// ---- DUTs/IO/PDOs/Outputs_B00B49A9.TcDUT
{attribute addProperty BoxType "EK1960-0000-0019"}
{attribute addProperty Id "Module_1_Channel_1_Standard_Output_X5_1AT %Q*BOOL811Module_1_Channel_2_Standard_Output_X5_2AT %Q*BOOL812Module_1_Channel_3_Standard_Output_X5_3AT %Q*BOOL813Module_1_Channel_4_Standard_Output_X5_4AT %Q*BOOL814Module_2_Channel_1_Standard_Output_X5_5AT %Q*BOOL811Module_2_Channel_2_Standard_Output_X5_6AT %Q*BOOL812Module_2_Channel_3_Standard_Output_X5_7AT %Q*BOOL813Module_2_Channel_4_Standard_Output_X5_8AT %Q*BOOL814Module_3_Channel_1_Standard_Output_X7_1AT %Q*BOOL811Module_3_Channel_2_Standard_Output_X7_2AT %Q*BOOL812Module_3_Channel_3_Standard_Output_X7_3AT %Q*BOOL813Module_3_Channel_4_Standard_Output_X7_4AT %Q*BOOL814Module_4_Channel_1_Standard_Output_X7_5AT %Q*BOOL811Module_4_Channel_2_Standard_Output_X7_6AT %Q*BOOL812Module_4_Channel_3_Standard_Output_X7_7AT %Q*BOOL813Module_4_Channel_4_Standard_Output_X7_8AT %Q*BOOL814Module_5_Channel_1_Standard_Output_X9_1AT %Q*BOOL811Module_5_Channel_2_Standard_Output_X9_2AT %Q*BOOL812Module_5_Channel_3_Standard_Output_X9_3AT %Q*BOOL813Module_5_Channel_4_Standard_Output_X9_4AT %Q*BOOL814Module_6_Channel_1_Standard_Output_X9_5AT %Q*BOOL811Module_6_Channel_2_Standard_Output_X9_6AT %Q*BOOL812Module_6_Channel_3_Standard_Output_X9_7AT %Q*BOOL813Module_6_Channel_4_Standard_Output_X9_8AT %Q*BOOL814Relais_Module_Channel_1_Standard_Output_X4_1_X4_5AT %Q*BOOL811Relais_Module_Channel_2_Standard_Output_X4_2_X4_6AT %Q*BOOL812Relais_Module_Channel_3_Standard_Output_X4_3_X4_7AT %Q*BOOL813Relais_Module_Channel_4_Standard_Output_X4_4_X4_8AT %Q*BOOL814"}
{attribute addProperty CRC "2953529769"}
{attribute addProperty SizeInBites "224"}
{attribute addProperty SizeInBytes "28"}
TYPE Outputs_B00B49A9 :
STRUCT
	{attribute addProperty Name "Module_1_Channel_1_Standard_Output_X5_1"}
	Module_1_Channel_1_Standard_Output_X5_1 AT %Q* : BOOL;
	{attribute addProperty Name "Module_1_Channel_2_Standard_Output_X5_2"}
	Module_1_Channel_2_Standard_Output_X5_2 AT %Q* : BOOL;
	{attribute addProperty Name "Module_1_Channel_3_Standard_Output_X5_3"}
	Module_1_Channel_3_Standard_Output_X5_3 AT %Q* : BOOL;
	{attribute addProperty Name "Module_1_Channel_4_Standard_Output_X5_4"}
	Module_1_Channel_4_Standard_Output_X5_4 AT %Q* : BOOL;
	{attribute addProperty Name "Module_2_Channel_1_Standard_Output_X5_5"}
	Module_2_Channel_1_Standard_Output_X5_5 AT %Q* : BOOL;
	{attribute addProperty Name "Module_2_Channel_2_Standard_Output_X5_6"}
	Module_2_Channel_2_Standard_Output_X5_6 AT %Q* : BOOL;
	{attribute addProperty Name "Module_2_Channel_3_Standard_Output_X5_7"}
	Module_2_Channel_3_Standard_Output_X5_7 AT %Q* : BOOL;
	{attribute addProperty Name "Module_2_Channel_4_Standard_Output_X5_8"}
	Module_2_Channel_4_Standard_Output_X5_8 AT %Q* : BOOL;
	{attribute addProperty Name "Module_3_Channel_1_Standard_Output_X7_1"}
	Module_3_Channel_1_Standard_Output_X7_1 AT %Q* : BOOL;
	{attribute addProperty Name "Module_3_Channel_2_Standard_Output_X7_2"}
	Module_3_Channel_2_Standard_Output_X7_2 AT %Q* : BOOL;
	{attribute addProperty Name "Module_3_Channel_3_Standard_Output_X7_3"}
	Module_3_Channel_3_Standard_Output_X7_3 AT %Q* : BOOL;
	{attribute addProperty Name "Module_3_Channel_4_Standard_Output_X7_4"}
	Module_3_Channel_4_Standard_Output_X7_4 AT %Q* : BOOL;
	{attribute addProperty Name "Module_4_Channel_1_Standard_Output_X7_5"}
	Module_4_Channel_1_Standard_Output_X7_5 AT %Q* : BOOL;
	{attribute addProperty Name "Module_4_Channel_2_Standard_Output_X7_6"}
	Module_4_Channel_2_Standard_Output_X7_6 AT %Q* : BOOL;
	{attribute addProperty Name "Module_4_Channel_3_Standard_Output_X7_7"}
	Module_4_Channel_3_Standard_Output_X7_7 AT %Q* : BOOL;
	{attribute addProperty Name "Module_4_Channel_4_Standard_Output_X7_8"}
	Module_4_Channel_4_Standard_Output_X7_8 AT %Q* : BOOL;
	{attribute addProperty Name "Module_5_Channel_1_Standard_Output_X9_1"}
	Module_5_Channel_1_Standard_Output_X9_1 AT %Q* : BOOL;
	{attribute addProperty Name "Module_5_Channel_2_Standard_Output_X9_2"}
	Module_5_Channel_2_Standard_Output_X9_2 AT %Q* : BOOL;
	{attribute addProperty Name "Module_5_Channel_3_Standard_Output_X9_3"}
	Module_5_Channel_3_Standard_Output_X9_3 AT %Q* : BOOL;
	{attribute addProperty Name "Module_5_Channel_4_Standard_Output_X9_4"}
	Module_5_Channel_4_Standard_Output_X9_4 AT %Q* : BOOL;
	{attribute addProperty Name "Module_6_Channel_1_Standard_Output_X9_5"}
	Module_6_Channel_1_Standard_Output_X9_5 AT %Q* : BOOL;
	{attribute addProperty Name "Module_6_Channel_2_Standard_Output_X9_6"}
	Module_6_Channel_2_Standard_Output_X9_6 AT %Q* : BOOL;
	{attribute addProperty Name "Module_6_Channel_3_Standard_Output_X9_7"}
	Module_6_Channel_3_Standard_Output_X9_7 AT %Q* : BOOL;
	{attribute addProperty Name "Module_6_Channel_4_Standard_Output_X9_8"}
	Module_6_Channel_4_Standard_Output_X9_8 AT %Q* : BOOL;
	{attribute addProperty Name "Relais_Module_Channel_1_Standard_Output_X4_1_X4_5"}
	Relais_Module_Channel_1_Standard_Output_X4_1_X4_5 AT %Q* : BOOL;
	{attribute addProperty Name "Relais_Module_Channel_2_Standard_Output_X4_2_X4_6"}
	Relais_Module_Channel_2_Standard_Output_X4_2_X4_6 AT %Q* : BOOL;
	{attribute addProperty Name "Relais_Module_Channel_3_Standard_Output_X4_3_X4_7"}
	Relais_Module_Channel_3_Standard_Output_X4_3_X4_7 AT %Q* : BOOL;
	{attribute addProperty Name "Relais_Module_Channel_4_Standard_Output_X4_4_X4_8"}
	Relais_Module_Channel_4_Standard_Output_X4_4_X4_8 AT %Q* : BOOL;
END_STRUCT
END_TYPE

// ---- DUTs/IO/PDOs/Module_1_FSoE_DD00D81F.TcDUT
{attribute addProperty BoxType "EK1960-0000-0019"}
{attribute addProperty Id "FSoE_InputsFSoE_Inputs_FED5CD6512015FSoE_OutputsFSoE_Outputs_931DC9C512015"}
{attribute addProperty CRC "3707820063"}
{attribute addProperty SizeInBites "240"}
{attribute addProperty SizeInBytes "30"}
TYPE Module_1_FSoE_DD00D81F :
STRUCT
	{attribute addProperty Name "FSoE_Inputs"}
	FSoE_Inputs  : FSoE_Inputs_FED5CD65;
	{attribute addProperty Name "FSoE_Outputs"}
	FSoE_Outputs  : FSoE_Outputs_931DC9C5;
END_STRUCT
END_TYPE

// ---- DUTs/IO/PDOs/Module_2_FSOUT_3AD10D8E.TcDUT
{attribute addProperty BoxType "EK1960-0000-0019"}
{attribute addProperty Id "OutputsOutputs_B00B49A922428"}
{attribute addProperty CRC "986779022"}
{attribute addProperty SizeInBites "224"}
{attribute addProperty SizeInBytes "28"}
TYPE Module_2_FSOUT_3AD10D8E :
STRUCT
	{attribute addProperty Name "Outputs"}
	Outputs  : Outputs_B00B49A9;
END_STRUCT
END_TYPE

// ---- DUTs/IO/PDOs/FSoE_Inputs_91F6EA71.TcDUT
{attribute addProperty BoxType "EK1960-0000-0021"}
{attribute addProperty Id "FSOEAT %I*FSOE_320A0AF812015"}
{attribute addProperty CRC "2448878193"}
{attribute addProperty SizeInBites "120"}
{attribute addProperty SizeInBytes "15"}
TYPE FSoE_Inputs_91F6EA71 :
STRUCT
	{attribute addProperty Name "FSOE"}
	FSOE AT %I* : FSOE_320A0AF8;
END_STRUCT
END_TYPE

// ---- DUTs/IO/PDOs/FSoE_Outputs_DB0FA8F7.TcDUT
{attribute addProperty BoxType "EK1960-0000-0021"}
{attribute addProperty Id "FSOEAT %Q*FSOE_B358BD5C12015"}
{attribute addProperty CRC "3675236599"}
{attribute addProperty SizeInBites "120"}
{attribute addProperty SizeInBytes "15"}
TYPE FSoE_Outputs_DB0FA8F7 :
STRUCT
	{attribute addProperty Name "FSOE"}
	FSOE AT %Q* : FSOE_B358BD5C;
END_STRUCT
END_TYPE

// ---- DUTs/IO/PDOs/Outputs_5BA3BA9A.TcDUT
{attribute addProperty BoxType "EK1960-0000-0021"}
{attribute addProperty Id "Module_1_Channel_1_Standard_Output_X5_1AT %Q*BOOL811Module_1_Channel_2_Standard_Output_X5_2AT %Q*BOOL812Module_1_Channel_3_Standard_Output_X5_3AT %Q*BOOL813Module_1_Channel_4_Standard_Output_X5_4AT %Q*BOOL814Module_2_Channel_1_Standard_Output_X5_5AT %Q*BOOL811Module_2_Channel_2_Standard_Output_X5_6AT %Q*BOOL812Module_2_Channel_3_Standard_Output_X5_7AT %Q*BOOL813Module_2_Channel_4_Standard_Output_X5_8AT %Q*BOOL814Module_3_Channel_1_Standard_Output_X7_1AT %Q*BOOL811Module_3_Channel_2_Standard_Output_X7_2AT %Q*BOOL812Module_3_Channel_3_Standard_Output_X7_3AT %Q*BOOL813Module_3_Channel_4_Standard_Output_X7_4AT %Q*BOOL814Module_4_Channel_1_Standard_Output_X7_5AT %Q*BOOL811Module_4_Channel_2_Standard_Output_X7_6AT %Q*BOOL812Module_4_Channel_3_Standard_Output_X7_7AT %Q*BOOL813Module_4_Channel_4_Standard_Output_X7_8AT %Q*BOOL814Module_5_Channel_1_Standard_Output_X9_1AT %Q*BOOL811Module_5_Channel_2_Standard_Output_X9_2AT %Q*BOOL812Module_5_Channel_3_Standard_Output_X9_3AT %Q*BOOL813Module_5_Channel_4_Standard_Output_X9_4AT %Q*BOOL814Module_6_Channel_1_Standard_Output_X9_5AT %Q*BOOL811Module_6_Channel_2_Standard_Output_X9_6AT %Q*BOOL812Module_6_Channel_3_Standard_Output_X9_7AT %Q*BOOL813Module_6_Channel_4_Standard_Output_X9_8AT %Q*BOOL814"}
{attribute addProperty CRC "1537456794"}
{attribute addProperty SizeInBites "192"}
{attribute addProperty SizeInBytes "24"}
TYPE Outputs_5BA3BA9A :
STRUCT
	{attribute addProperty Name "Module_1_Channel_1_Standard_Output_X5_1"}
	Module_1_Channel_1_Standard_Output_X5_1 AT %Q* : BOOL;
	{attribute addProperty Name "Module_1_Channel_2_Standard_Output_X5_2"}
	Module_1_Channel_2_Standard_Output_X5_2 AT %Q* : BOOL;
	{attribute addProperty Name "Module_1_Channel_3_Standard_Output_X5_3"}
	Module_1_Channel_3_Standard_Output_X5_3 AT %Q* : BOOL;
	{attribute addProperty Name "Module_1_Channel_4_Standard_Output_X5_4"}
	Module_1_Channel_4_Standard_Output_X5_4 AT %Q* : BOOL;
	{attribute addProperty Name "Module_2_Channel_1_Standard_Output_X5_5"}
	Module_2_Channel_1_Standard_Output_X5_5 AT %Q* : BOOL;
	{attribute addProperty Name "Module_2_Channel_2_Standard_Output_X5_6"}
	Module_2_Channel_2_Standard_Output_X5_6 AT %Q* : BOOL;
	{attribute addProperty Name "Module_2_Channel_3_Standard_Output_X5_7"}
	Module_2_Channel_3_Standard_Output_X5_7 AT %Q* : BOOL;
	{attribute addProperty Name "Module_2_Channel_4_Standard_Output_X5_8"}
	Module_2_Channel_4_Standard_Output_X5_8 AT %Q* : BOOL;
	{attribute addProperty Name "Module_3_Channel_1_Standard_Output_X7_1"}
	Module_3_Channel_1_Standard_Output_X7_1 AT %Q* : BOOL;
	{attribute addProperty Name "Module_3_Channel_2_Standard_Output_X7_2"}
	Module_3_Channel_2_Standard_Output_X7_2 AT %Q* : BOOL;
	{attribute addProperty Name "Module_3_Channel_3_Standard_Output_X7_3"}
	Module_3_Channel_3_Standard_Output_X7_3 AT %Q* : BOOL;
	{attribute addProperty Name "Module_3_Channel_4_Standard_Output_X7_4"}
	Module_3_Channel_4_Standard_Output_X7_4 AT %Q* : BOOL;
	{attribute addProperty Name "Module_4_Channel_1_Standard_Output_X7_5"}
	Module_4_Channel_1_Standard_Output_X7_5 AT %Q* : BOOL;
	{attribute addProperty Name "Module_4_Channel_2_Standard_Output_X7_6"}
	Module_4_Channel_2_Standard_Output_X7_6 AT %Q* : BOOL;
	{attribute addProperty Name "Module_4_Channel_3_Standard_Output_X7_7"}
	Module_4_Channel_3_Standard_Output_X7_7 AT %Q* : BOOL;
	{attribute addProperty Name "Module_4_Channel_4_Standard_Output_X7_8"}
	Module_4_Channel_4_Standard_Output_X7_8 AT %Q* : BOOL;
	{attribute addProperty Name "Module_5_Channel_1_Standard_Output_X9_1"}
	Module_5_Channel_1_Standard_Output_X9_1 AT %Q* : BOOL;
	{attribute addProperty Name "Module_5_Channel_2_Standard_Output_X9_2"}
	Module_5_Channel_2_Standard_Output_X9_2 AT %Q* : BOOL;
	{attribute addProperty Name "Module_5_Channel_3_Standard_Output_X9_3"}
	Module_5_Channel_3_Standard_Output_X9_3 AT %Q* : BOOL;
	{attribute addProperty Name "Module_5_Channel_4_Standard_Output_X9_4"}
	Module_5_Channel_4_Standard_Output_X9_4 AT %Q* : BOOL;
	{attribute addProperty Name "Module_6_Channel_1_Standard_Output_X9_5"}
	Module_6_Channel_1_Standard_Output_X9_5 AT %Q* : BOOL;
	{attribute addProperty Name "Module_6_Channel_2_Standard_Output_X9_6"}
	Module_6_Channel_2_Standard_Output_X9_6 AT %Q* : BOOL;
	{attribute addProperty Name "Module_6_Channel_3_Standard_Output_X9_7"}
	Module_6_Channel_3_Standard_Output_X9_7 AT %Q* : BOOL;
	{attribute addProperty Name "Module_6_Channel_4_Standard_Output_X9_8"}
	Module_6_Channel_4_Standard_Output_X9_8 AT %Q* : BOOL;
END_STRUCT
END_TYPE

// ---- DUTs/IO/PDOs/Module_1_FSoE_DA01C73E.TcDUT
{attribute addProperty BoxType "EK1960-0000-0021"}
{attribute addProperty Id "FSoE_InputsFSoE_Inputs_91F6EA7112015FSoE_OutputsFSoE_Outputs_DB0FA8F712015"}
{attribute addProperty CRC "3657549630"}
{attribute addProperty SizeInBites "240"}
{attribute addProperty SizeInBytes "30"}
TYPE Module_1_FSoE_DA01C73E :
STRUCT
	{attribute addProperty Name "FSoE_Inputs"}
	FSoE_Inputs  : FSoE_Inputs_91F6EA71;
	{attribute addProperty Name "FSoE_Outputs"}
	FSoE_Outputs  : FSoE_Outputs_DB0FA8F7;
END_STRUCT
END_TYPE

// ---- DUTs/IO/PDOs/Module_2_FSOUT_9F3624CE.TcDUT
{attribute addProperty BoxType "EK1960-0000-0021"}
{attribute addProperty Id "OutputsOutputs_5BA3BA9A19224"}
{attribute addProperty CRC "2671125710"}
{attribute addProperty SizeInBites "192"}
{attribute addProperty SizeInBytes "24"}
TYPE Module_2_FSOUT_9F3624CE :
STRUCT
	{attribute addProperty Name "Outputs"}
	Outputs  : Outputs_5BA3BA9A;
END_STRUCT
END_TYPE

// ---- DUTs/IO/PDOs/FSoE_Inputs_0C161FF7.TcDUT
{attribute addProperty BoxType "EK1960-2600-0019"}
{attribute addProperty Id "FSOEAT %I*FSOE_704ED52312015"}
{attribute addProperty CRC "202776567"}
{attribute addProperty SizeInBites "120"}
{attribute addProperty SizeInBytes "15"}
TYPE FSoE_Inputs_0C161FF7 :
STRUCT
	{attribute addProperty Name "FSOE"}
	FSOE AT %I* : FSOE_704ED523;
END_STRUCT
END_TYPE

// ---- DUTs/IO/PDOs/FSoE_Outputs_E86FAAD6.TcDUT
{attribute addProperty BoxType "EK1960-2600-0019"}
{attribute addProperty Id "FSOEAT %Q*FSOE_340991D312015"}
{attribute addProperty CRC "3899632342"}
{attribute addProperty SizeInBites "120"}
{attribute addProperty SizeInBytes "15"}
TYPE FSoE_Outputs_E86FAAD6 :
STRUCT
	{attribute addProperty Name "FSOE"}
	FSOE AT %Q* : FSOE_340991D3;
END_STRUCT
END_TYPE

// ---- DUTs/IO/PDOs/Module_1_FSoE_DA1FCD51.TcDUT
{attribute addProperty BoxType "EK1960-2600-0019"}
{attribute addProperty Id "FSoE_InputsFSoE_Inputs_0C161FF712015FSoE_OutputsFSoE_Outputs_E86FAAD612015"}
{attribute addProperty CRC "3659517265"}
{attribute addProperty SizeInBites "240"}
{attribute addProperty SizeInBytes "30"}
TYPE Module_1_FSoE_DA1FCD51 :
STRUCT
	{attribute addProperty Name "FSoE_Inputs"}
	FSoE_Inputs  : FSoE_Inputs_0C161FF7;
	{attribute addProperty Name "FSoE_Outputs"}
	FSoE_Outputs  : FSoE_Outputs_E86FAAD6;
END_STRUCT
END_TYPE

// ---- DUTs/IO/PDOs/FSoE_Inputs_CBB11F24.TcDUT
{attribute addProperty BoxType "EK1960-2600-0021"}
{attribute addProperty Id "FSOEAT %I*FSOE_3B47B0C112015"}
{attribute addProperty CRC "3417382692"}
{attribute addProperty SizeInBites "120"}
{attribute addProperty SizeInBytes "15"}
TYPE FSoE_Inputs_CBB11F24 :
STRUCT
	{attribute addProperty Name "FSOE"}
	FSOE AT %I* : FSOE_3B47B0C1;
END_STRUCT
END_TYPE

// ---- DUTs/IO/PDOs/FSoE_Outputs_616B4B11.TcDUT
{attribute addProperty BoxType "EK1960-2600-0021"}
{attribute addProperty Id "FSOEAT %Q*FSOE_9F05737212015"}
{attribute addProperty CRC "1634421521"}
{attribute addProperty SizeInBites "120"}
{attribute addProperty SizeInBytes "15"}
TYPE FSoE_Outputs_616B4B11 :
STRUCT
	{attribute addProperty Name "FSOE"}
	FSOE AT %Q* : FSOE_9F057372;
END_STRUCT
END_TYPE

// ---- DUTs/IO/PDOs/Module_1_FSoE_1C2EAE46.TcDUT
{attribute addProperty BoxType "EK1960-2600-0021"}
{attribute addProperty Id "FSoE_InputsFSoE_Inputs_CBB11F2412015FSoE_OutputsFSoE_Outputs_616B4B1112015"}
{attribute addProperty CRC "472821318"}
{attribute addProperty SizeInBites "240"}
{attribute addProperty SizeInBytes "30"}
TYPE Module_1_FSoE_1C2EAE46 :
STRUCT
	{attribute addProperty Name "FSoE_Inputs"}
	FSoE_Inputs  : FSoE_Inputs_CBB11F24;
	{attribute addProperty Name "FSoE_Outputs"}
	FSoE_Outputs  : FSoE_Outputs_616B4B11;
END_STRUCT
END_TYPE

// ---- DUTs/IO/Boxes/EK1100_179A0949.TcDUT
{attribute addProperty BoxType "EK1100-0000-0018"}
{attribute addProperty Id "InfoDataInfoData_192954DE162"}
{attribute addProperty CRC "395970889"}
{attribute addProperty SizeInBites "16"}
{attribute addProperty SizeInBytes "2"}
TYPE EK1100_179A0949 :
STRUCT
	{attribute addProperty Name "InfoData"}
	InfoData : InfoData_192954DE;
END_STRUCT
END_TYPE

// ---- DUTs/IO/Boxes/EK1122_179A0949.TcDUT
{attribute addProperty BoxType "EK1122-0000-0018"}
{attribute addProperty Id "InfoDataInfoData_192954DE162"}
{attribute addProperty CRC "395970889"}
{attribute addProperty SizeInBites "16"}
{attribute addProperty SizeInBytes "2"}
TYPE EK1122_179A0949 :
STRUCT
	{attribute addProperty Name "InfoData"}
	InfoData : InfoData_192954DE;
END_STRUCT
END_TYPE

// ---- DUTs/IO/Boxes/EJ1100_179A0949.TcDUT
{attribute addProperty BoxType "EJ1100-0000-0018"}
{attribute addProperty Id "InfoDataInfoData_192954DE162"}
{attribute addProperty CRC "395970889"}
{attribute addProperty SizeInBites "16"}
{attribute addProperty SizeInBytes "2"}
TYPE EJ1100_179A0949 :
STRUCT
	{attribute addProperty Name "InfoData"}
	InfoData : InfoData_192954DE;
END_STRUCT
END_TYPE

// ---- DUTs/IO/Boxes/EJ1101_6969C224.TcDUT
{attribute addProperty BoxType "EJ1101-0022-0016"}
{attribute addProperty Id "WcStateAT %I*WcState_28A8677510.1250InfoDataAT %I*InfoData_BC63D37F80100"}
{attribute addProperty CRC "752626490"}
{attribute addProperty SizeInBites "81"}
{attribute addProperty SizeInBytes "10.125"}
TYPE EJ1101_6969C224 :
STRUCT
	{attribute addProperty Name "WcState"}
	WcState : WcState_28A86775;
	{attribute addProperty Name "InfoData"}
	InfoData : InfoData_BC63D37F;
END_STRUCT
END_TYPE

// ---- DUTs/IO/Boxes/EJ1008_772BB414.TcDUT
{attribute addProperty BoxType "EJ1008-0000-0017"}
{attribute addProperty Id "ChannelAT %I*ARRAY[0..7] OF Channel_E4AEF59E6480WcStateAT %I*WcState_98A4DF7520.250InfoDataAT %I*InfoData_192954DE1620"}
{attribute addProperty CRC "2007808796"}
{attribute addProperty SizeInBites "82"}
{attribute addProperty SizeInBytes "10.25"}
TYPE EJ1008_772BB414 :
STRUCT
	{attribute addProperty Name "Channel"}
	Channel : ARRAY[0..7] OF Channel_E4AEF59E;
	{attribute addProperty Name "WcState"}
	WcState : WcState_98A4DF75;
	{attribute addProperty Name "InfoData"}
	InfoData : InfoData_192954DE;
END_STRUCT
END_TYPE

// ---- DUTs/IO/Boxes/EJ1128_772BB414.TcDUT
{attribute addProperty BoxType "EJ1128-0000-0016"}
{attribute addProperty Id "ChannelAT %I*ARRAY[0..7] OF Channel_E4AEF59E6480WcStateAT %I*WcState_98A4DF7520.250InfoDataAT %I*InfoData_192954DE1620"}
{attribute addProperty CRC "2007808796"}
{attribute addProperty SizeInBites "82"}
{attribute addProperty SizeInBytes "10.25"}
TYPE EJ1128_772BB414 :
STRUCT
	{attribute addProperty Name "Channel"}
	Channel : ARRAY[0..7] OF Channel_E4AEF59E;
	{attribute addProperty Name "WcState"}
	WcState : WcState_98A4DF75;
	{attribute addProperty Name "InfoData"}
	InfoData : InfoData_192954DE;
END_STRUCT
END_TYPE

// ---- DUTs/IO/Boxes/EJ1809_248EAA34.TcDUT
{attribute addProperty BoxType "EJ1809-0000-0017"}
{attribute addProperty Id "ChannelAT %I*ARRAY[0..15] OF Channel_E4AEF59E128160WcStateAT %I*WcState_98A4DF7520.250InfoDataAT %I*InfoData_192954DE1620"}
{attribute addProperty CRC "4206052659"}
{attribute addProperty SizeInBites "146"}
{attribute addProperty SizeInBytes "18.25"}
TYPE EJ1809_248EAA34 :
STRUCT
	{attribute addProperty Name "Channel"}
	Channel : ARRAY[0..15] OF Channel_E4AEF59E;
	{attribute addProperty Name "WcState"}
	WcState : WcState_98A4DF75;
	{attribute addProperty Name "InfoData"}
	InfoData : InfoData_192954DE;
END_STRUCT
END_TYPE

// ---- DUTs/IO/Boxes/EJ1819_248EAA34.TcDUT
{attribute addProperty BoxType "EJ1819-0000-0017"}
{attribute addProperty Id "ChannelAT %I*ARRAY[0..15] OF Channel_E4AEF59E128160WcStateAT %I*WcState_98A4DF7520.250InfoDataAT %I*InfoData_192954DE1620"}
{attribute addProperty CRC "4206052659"}
{attribute addProperty SizeInBites "146"}
{attribute addProperty SizeInBytes "18.25"}
TYPE EJ1819_248EAA34 :
STRUCT
	{attribute addProperty Name "Channel"}
	Channel : ARRAY[0..15] OF Channel_E4AEF59E;
	{attribute addProperty Name "WcState"}
	WcState : WcState_98A4DF75;
	{attribute addProperty Name "InfoData"}
	InfoData : InfoData_192954DE;
END_STRUCT
END_TYPE

// ---- DUTs/IO/Boxes/EJ1859_538B459D.TcDUT
{attribute addProperty BoxType "EJ1859-0000-0017"}
{attribute addProperty Id "ChannelAT %I*ARRAY[0..7] OF Channel_E4AEF59E6480Channel_1AT %Q*ARRAY[0..7] OF Channel_7F374EB06480WcStateAT %I*WcState_98A4DF7520.250InfoDataAT %I*InfoData_192954DE1620"}
{attribute addProperty CRC "4038043443"}
{attribute addProperty SizeInBites "146"}
{attribute addProperty SizeInBytes "18.25"}
TYPE EJ1859_538B459D :
STRUCT
	{attribute addProperty Name "Channel"}
	Channel : ARRAY[0..7] OF Channel_E4AEF59E;
	{attribute addProperty Name "Channel_1"}
	Channel_1 : ARRAY[0..7] OF Channel_7F374EB0;
	{attribute addProperty Name "WcState"}
	WcState : WcState_98A4DF75;
	{attribute addProperty Name "InfoData"}
	InfoData : InfoData_192954DE;
END_STRUCT
END_TYPE

// ---- DUTs/IO/Boxes/EJ1889_248EAA34.TcDUT
{attribute addProperty BoxType "EJ1889-0000-0017"}
{attribute addProperty Id "ChannelAT %I*ARRAY[0..15] OF Channel_E4AEF59E128160WcStateAT %I*WcState_98A4DF7520.250InfoDataAT %I*InfoData_192954DE1620"}
{attribute addProperty CRC "4206052659"}
{attribute addProperty SizeInBites "146"}
{attribute addProperty SizeInBytes "18.25"}
TYPE EJ1889_248EAA34 :
STRUCT
	{attribute addProperty Name "Channel"}
	Channel : ARRAY[0..15] OF Channel_E4AEF59E;
	{attribute addProperty Name "WcState"}
	WcState : WcState_98A4DF75;
	{attribute addProperty Name "InfoData"}
	InfoData : InfoData_192954DE;
END_STRUCT
END_TYPE

// ---- DUTs/IO/Boxes/EJ1122_179A0949.TcDUT
{attribute addProperty BoxType "EJ1122-0000-0016"}
{attribute addProperty Id "InfoDataInfoData_192954DE162"}
{attribute addProperty CRC "395970889"}
{attribute addProperty SizeInBites "16"}
{attribute addProperty SizeInBytes "2"}
TYPE EJ1122_179A0949 :
STRUCT
	{attribute addProperty Name "InfoData"}
	InfoData : InfoData_192954DE;
END_STRUCT
END_TYPE

// ---- DUTs/IO/Boxes/EJ2008_A854BE6D.TcDUT
{attribute addProperty BoxType "EJ2008-0000-0017"}
{attribute addProperty Id "ChannelAT %Q*ARRAY[0..7] OF Channel_7F374EB06480WcStateAT %I*WcState_28A8677510.1250InfoDataAT %I*InfoData_192954DE1620"}
{attribute addProperty CRC "1482585628"}
{attribute addProperty SizeInBites "81"}
{attribute addProperty SizeInBytes "10.125"}
TYPE EJ2008_A854BE6D :
STRUCT
	{attribute addProperty Name "Channel"}
	Channel : ARRAY[0..7] OF Channel_7F374EB0;
	{attribute addProperty Name "WcState"}
	WcState : WcState_28A86775;
	{attribute addProperty Name "InfoData"}
	InfoData : InfoData_192954DE;
END_STRUCT
END_TYPE

// ---- DUTs/IO/Boxes/EJ2128_A854BE6D.TcDUT
{attribute addProperty BoxType "EJ2128-0000-0016"}
{attribute addProperty Id "ChannelAT %Q*ARRAY[0..7] OF Channel_7F374EB06480WcStateAT %I*WcState_28A8677510.1250InfoDataAT %I*InfoData_192954DE1620"}
{attribute addProperty CRC "1482585628"}
{attribute addProperty SizeInBites "81"}
{attribute addProperty SizeInBytes "10.125"}
TYPE EJ2128_A854BE6D :
STRUCT
	{attribute addProperty Name "Channel"}
	Channel : ARRAY[0..7] OF Channel_7F374EB0;
	{attribute addProperty Name "WcState"}
	WcState : WcState_28A86775;
	{attribute addProperty Name "InfoData"}
	InfoData : InfoData_192954DE;
END_STRUCT
END_TYPE

// ---- DUTs/IO/Boxes/EJ2502_68F74D5A.TcDUT
{attribute addProperty BoxType "EJ2502-0000-0023"}
{attribute addProperty Id "PWM_Outputs_ChannelAT %Q*ARRAY[0..1] OF PWM_Outputs_Channel_A83D42AA3240WcStateAT %I*WcState_28A8677510.1250InfoDataAT %I*InfoData_BC63D37F80100"}
{attribute addProperty CRC "1493002450"}
{attribute addProperty SizeInBites "113"}
{attribute addProperty SizeInBytes "14.125"}
TYPE EJ2502_68F74D5A :
STRUCT
	{attribute addProperty Name "PWM_Outputs_Channel"}
	PWM_Outputs_Channel : ARRAY[0..1] OF PWM_Outputs_Channel_A83D42AA;
	{attribute addProperty Name "WcState"}
	WcState : WcState_28A86775;
	{attribute addProperty Name "InfoData"}
	InfoData : InfoData_BC63D37F;
END_STRUCT
END_TYPE

// ---- DUTs/IO/Boxes/EJ2521_A10F5EEB.TcDUT
{attribute addProperty BoxType "EJ2521-0224-0016"}
{attribute addProperty Id "PTO_StatusAT %I*PTO_Status_B9BB57FE1620ENC_Status_compactAT %I*ENC_Status_compact_FA080ECA4860PLS_Status_ChannelAT %I*ARRAY[0..1] OF PLS_Status_Channel_7A2392D13240PTO_ControlAT %Q*PTO_Control_0A6210C33240PTO_Target_compactAT %Q*PTO_Target_compact_C80C22BB1620ENC_Control_compactAT %Q*ENC_Control_compact_5C86AA9D3240PLS_Control_compact_ChannelAT %Q*ARRAY[0..3] OF PLS_Control_compact_Channel_F7E9C67496120WcStateAT %I*WcState_98A4DF7520.250InfoDataAT %I*InfoData_BC63D37F80100"}
{attribute addProperty CRC "3307808944"}
{attribute addProperty SizeInBites "354"}
{attribute addProperty SizeInBytes "44.25"}
TYPE EJ2521_A10F5EEB :
STRUCT
	{attribute addProperty Name "PTO_Status"}
	PTO_Status : PTO_Status_B9BB57FE;
	{attribute addProperty Name "ENC_Status_compact"}
	ENC_Status_compact : ENC_Status_compact_FA080ECA;
	{attribute addProperty Name "PLS_Status_Channel"}
	PLS_Status_Channel : ARRAY[0..1] OF PLS_Status_Channel_7A2392D1;
	{attribute addProperty Name "PTO_Control"}
	PTO_Control : PTO_Control_0A6210C3;
	{attribute addProperty Name "PTO_Target_compact"}
	PTO_Target_compact : PTO_Target_compact_C80C22BB;
	{attribute addProperty Name "ENC_Control_compact"}
	ENC_Control_compact : ENC_Control_compact_5C86AA9D;
	{attribute addProperty Name "PLS_Control_compact_Channel"}
	PLS_Control_compact_Channel : ARRAY[0..3] OF PLS_Control_compact_Channel_F7E9C674;
	{attribute addProperty Name "WcState"}
	WcState : WcState_98A4DF75;
	{attribute addProperty Name "InfoData"}
	InfoData : InfoData_BC63D37F;
END_STRUCT
END_TYPE

// ---- DUTs/IO/Boxes/EJ2522_58A1BC1F.TcDUT
{attribute addProperty BoxType "EJ2522-0000-0022"}
{attribute addProperty Id "PTO_Status_ChannelAT %I*ARRAY[0..1] OF PTO_Status_Channel_B9BB57FE3240ENC_Status_ChannelAT %I*ARRAY[0..2] OF ENC_Status_Channel_D7F8917396120PTO_Control_Channel_1AT %Q*PTO_Control_Channel_0A6210C33240PTO_Target_Channel_1AT %Q*PTO_Target_Channel_3945899C3240PTO_Control_Channel_2AT %Q*PTO_Control_Channel_0A6210C33240PTO_Target_Channel_2AT %Q*PTO_Target_Channel_3945899C3240ENC_Control_ChannelAT %Q*ARRAY[0..2] OF ENC_Control_Channel_8309D56E96120WcStateAT %I*WcState_98A4DF7520.250InfoDataAT %I*InfoData_BC63D37F80100"}
{attribute addProperty CRC "1184876195"}
{attribute addProperty SizeInBites "434"}
{attribute addProperty SizeInBytes "54.25"}
TYPE EJ2522_58A1BC1F :
STRUCT
	{attribute addProperty Name "PTO_Status_Channel"}
	PTO_Status_Channel : ARRAY[0..1] OF PTO_Status_Channel_B9BB57FE;
	{attribute addProperty Name "ENC_Status_Channel"}
	ENC_Status_Channel : ARRAY[0..2] OF ENC_Status_Channel_D7F89173;
	{attribute addProperty Name "PTO_Control_Channel_1"}
	PTO_Control_Channel_1 : PTO_Control_Channel_0A6210C3;
	{attribute addProperty Name "PTO_Target_Channel_1"}
	PTO_Target_Channel_1 : PTO_Target_Channel_3945899C;
	{attribute addProperty Name "PTO_Control_Channel_2"}
	PTO_Control_Channel_2 : PTO_Control_Channel_0A6210C3;
	{attribute addProperty Name "PTO_Target_Channel_2"}
	PTO_Target_Channel_2 : PTO_Target_Channel_3945899C;
	{attribute addProperty Name "ENC_Control_Channel"}
	ENC_Control_Channel : ARRAY[0..2] OF ENC_Control_Channel_8309D56E;
	{attribute addProperty Name "WcState"}
	WcState : WcState_98A4DF75;
	{attribute addProperty Name "InfoData"}
	InfoData : InfoData_BC63D37F;
END_STRUCT
END_TYPE

// ---- DUTs/IO/Boxes/EJ2809_859F43D2.TcDUT
{attribute addProperty BoxType "EJ2809-0000-0017"}
{attribute addProperty Id "ChannelAT %Q*ARRAY[0..15] OF Channel_7F374EB0128160WcStateAT %I*WcState_28A8677510.1250InfoDataAT %I*InfoData_192954DE1620"}
{attribute addProperty CRC "924279498"}
{attribute addProperty SizeInBites "145"}
{attribute addProperty SizeInBytes "18.125"}
TYPE EJ2809_859F43D2 :
STRUCT
	{attribute addProperty Name "Channel"}
	Channel : ARRAY[0..15] OF Channel_7F374EB0;
	{attribute addProperty Name "WcState"}
	WcState : WcState_28A86775;
	{attribute addProperty Name "InfoData"}
	InfoData : InfoData_192954DE;
END_STRUCT
END_TYPE

// ---- DUTs/IO/Boxes/EJ2889_859F43D2.TcDUT
{attribute addProperty BoxType "EJ2889-0000-0016"}
{attribute addProperty Id "ChannelAT %Q*ARRAY[0..15] OF Channel_7F374EB0128160WcStateAT %I*WcState_28A8677510.1250InfoDataAT %I*InfoData_192954DE1620"}
{attribute addProperty CRC "924279498"}
{attribute addProperty SizeInBites "145"}
{attribute addProperty SizeInBytes "18.125"}
TYPE EJ2889_859F43D2 :
STRUCT
	{attribute addProperty Name "Channel"}
	Channel : ARRAY[0..15] OF Channel_7F374EB0;
	{attribute addProperty Name "WcState"}
	WcState : WcState_28A86775;
	{attribute addProperty Name "InfoData"}
	InfoData : InfoData_192954DE;
END_STRUCT
END_TYPE

// ---- DUTs/IO/Boxes/EJ3004_25122C20.TcDUT
{attribute addProperty BoxType "EJ3004-0000-0019"}
{attribute addProperty Id "AI_Standard_ChannelAT %I*ARRAY[0..6] OF AI_Standard_Channel_5763EEB9128160WcStateAT %I*WcState_98A4DF7520.250InfoDataAT %I*InfoData_BC63D37F80100"}
{attribute addProperty CRC "3504630615"}
{attribute addProperty SizeInBites "210"}
{attribute addProperty SizeInBytes "26.25"}
TYPE EJ3004_25122C20 :
STRUCT
	{attribute addProperty Name "AI_Standard_Channel"}
	AI_Standard_Channel : ARRAY[0..6] OF AI_Standard_Channel_5763EEB9;
	{attribute addProperty Name "WcState"}
	WcState : WcState_98A4DF75;
	{attribute addProperty Name "InfoData"}
	InfoData : InfoData_BC63D37F;
END_STRUCT
END_TYPE

// ---- DUTs/IO/Boxes/EJ3004_BB821456.TcDUT
{attribute addProperty BoxType "EJ3004-0000-0020"}
{attribute addProperty Id "AI_Standard_ChannelAT %I*ARRAY[0..6] OF AI_Standard_Channel_F16A160D128160WcStateAT %I*WcState_98A4DF7520.250InfoDataAT %I*InfoData_BC63D37F80100"}
{attribute addProperty CRC "4042565249"}
{attribute addProperty SizeInBites "210"}
{attribute addProperty SizeInBytes "26.25"}
TYPE EJ3004_BB821456 :
STRUCT
	{attribute addProperty Name "AI_Standard_Channel"}
	AI_Standard_Channel : ARRAY[0..6] OF AI_Standard_Channel_F16A160D;
	{attribute addProperty Name "WcState"}
	WcState : WcState_98A4DF75;
	{attribute addProperty Name "InfoData"}
	InfoData : InfoData_BC63D37F;
END_STRUCT
END_TYPE

// ---- DUTs/IO/Boxes/EJ3048_EA60A077.TcDUT
{attribute addProperty BoxType "EJ3048-0000-0020"}
{attribute addProperty Id "AI_Standard_ChannelAT %I*ARRAY[0..14] OF AI_Standard_Channel_F16A160D256320WcStateAT %I*WcState_98A4DF7520.250InfoDataAT %I*InfoData_BC63D37F80100"}
{attribute addProperty CRC "1252681791"}
{attribute addProperty SizeInBites "338"}
{attribute addProperty SizeInBytes "42.25"}
TYPE EJ3048_EA60A077 :
STRUCT
	{attribute addProperty Name "AI_Standard_Channel"}
	AI_Standard_Channel : ARRAY[0..14] OF AI_Standard_Channel_F16A160D;
	{attribute addProperty Name "WcState"}
	WcState : WcState_98A4DF75;
	{attribute addProperty Name "InfoData"}
	InfoData : InfoData_BC63D37F;
END_STRUCT
END_TYPE

// ---- DUTs/IO/Boxes/EJ3058_EA60A077.TcDUT
{attribute addProperty BoxType "EJ3058-0000-0020"}
{attribute addProperty Id "AI_Standard_ChannelAT %I*ARRAY[0..14] OF AI_Standard_Channel_F16A160D256320WcStateAT %I*WcState_98A4DF7520.250InfoDataAT %I*InfoData_BC63D37F80100"}
{attribute addProperty CRC "1252681791"}
{attribute addProperty SizeInBites "338"}
{attribute addProperty SizeInBytes "42.25"}
TYPE EJ3058_EA60A077 :
STRUCT
	{attribute addProperty Name "AI_Standard_Channel"}
	AI_Standard_Channel : ARRAY[0..14] OF AI_Standard_Channel_F16A160D;
	{attribute addProperty Name "WcState"}
	WcState : WcState_98A4DF75;
	{attribute addProperty Name "InfoData"}
	InfoData : InfoData_BC63D37F;
END_STRUCT
END_TYPE

// ---- DUTs/IO/Boxes/EJ3068_EA60A077.TcDUT
{attribute addProperty BoxType "EJ3068-0000-0020"}
{attribute addProperty Id "AI_Standard_ChannelAT %I*ARRAY[0..14] OF AI_Standard_Channel_F16A160D256320WcStateAT %I*WcState_98A4DF7520.250InfoDataAT %I*InfoData_BC63D37F80100"}
{attribute addProperty CRC "1252681791"}
{attribute addProperty SizeInBites "338"}
{attribute addProperty SizeInBytes "42.25"}
TYPE EJ3068_EA60A077 :
STRUCT
	{attribute addProperty Name "AI_Standard_Channel"}
	AI_Standard_Channel : ARRAY[0..14] OF AI_Standard_Channel_F16A160D;
	{attribute addProperty Name "WcState"}
	WcState : WcState_98A4DF75;
	{attribute addProperty Name "InfoData"}
	InfoData : InfoData_BC63D37F;
END_STRUCT
END_TYPE

// ---- DUTs/IO/Boxes/EJ3104_B7B53025.TcDUT
{attribute addProperty BoxType "EJ3104-0000-0019"}
{attribute addProperty Id "AI_Standard_ChannelAT %I*ARRAY[0..6] OF AI_Standard_Channel_087F71C7128160WcStateAT %I*WcState_98A4DF7520.250InfoDataAT %I*InfoData_BC63D37F80100"}
{attribute addProperty CRC "1733492472"}
{attribute addProperty SizeInBites "210"}
{attribute addProperty SizeInBytes "26.25"}
TYPE EJ3104_B7B53025 :
STRUCT
	{attribute addProperty Name "AI_Standard_Channel"}
	AI_Standard_Channel : ARRAY[0..6] OF AI_Standard_Channel_087F71C7;
	{attribute addProperty Name "WcState"}
	WcState : WcState_98A4DF75;
	{attribute addProperty Name "InfoData"}
	InfoData : InfoData_BC63D37F;
END_STRUCT
END_TYPE

// ---- DUTs/IO/Boxes/EJ3108_EA60A077.TcDUT
{attribute addProperty BoxType "EJ3108-0000-0017"}
{attribute addProperty Id "AI_Standard_ChannelAT %I*ARRAY[0..14] OF AI_Standard_Channel_F16A160D256320WcStateAT %I*WcState_98A4DF7520.250InfoDataAT %I*InfoData_BC63D37F80100"}
{attribute addProperty CRC "1252681791"}
{attribute addProperty SizeInBites "338"}
{attribute addProperty SizeInBytes "42.25"}
TYPE EJ3108_EA60A077 :
STRUCT
	{attribute addProperty Name "AI_Standard_Channel"}
	AI_Standard_Channel : ARRAY[0..14] OF AI_Standard_Channel_F16A160D;
	{attribute addProperty Name "WcState"}
	WcState : WcState_98A4DF75;
	{attribute addProperty Name "InfoData"}
	InfoData : InfoData_BC63D37F;
END_STRUCT
END_TYPE

// ---- DUTs/IO/Boxes/EJ3108_060F55FF.TcDUT
{attribute addProperty BoxType "EJ3108-0000-0018"}
{attribute addProperty Id "AI_Standard_ChannelAT %I*ARRAY[0..14] OF AI_Standard_Channel_087F71C7256320WcStateAT %I*WcState_98A4DF7520.250InfoDataAT %I*InfoData_BC63D37F80100"}
{attribute addProperty CRC "3708563526"}
{attribute addProperty SizeInBites "338"}
{attribute addProperty SizeInBytes "42.25"}
TYPE EJ3108_060F55FF :
STRUCT
	{attribute addProperty Name "AI_Standard_Channel"}
	AI_Standard_Channel : ARRAY[0..14] OF AI_Standard_Channel_087F71C7;
	{attribute addProperty Name "WcState"}
	WcState : WcState_98A4DF75;
	{attribute addProperty Name "InfoData"}
	InfoData : InfoData_BC63D37F;
END_STRUCT
END_TYPE

// ---- DUTs/IO/Boxes/EJ3202_559337F5.TcDUT
{attribute addProperty BoxType "EJ3202-0000-0019"}
{attribute addProperty Id "RTD_Inputs_ChannelAT %I*ARRAY[0..2] OF RTD_Inputs_Channel_5763EEB96480WcStateAT %I*WcState_98A4DF7520.250InfoDataAT %I*InfoData_BC63D37F80100"}
{attribute addProperty CRC "2714103225"}
{attribute addProperty SizeInBites "146"}
{attribute addProperty SizeInBytes "18.25"}
TYPE EJ3202_559337F5 :
STRUCT
	{attribute addProperty Name "RTD_Inputs_Channel"}
	RTD_Inputs_Channel : ARRAY[0..2] OF RTD_Inputs_Channel_5763EEB9;
	{attribute addProperty Name "WcState"}
	WcState : WcState_98A4DF75;
	{attribute addProperty Name "InfoData"}
	InfoData : InfoData_BC63D37F;
END_STRUCT
END_TYPE

// ---- DUTs/IO/Boxes/EJ3214_712ECA1B.TcDUT
{attribute addProperty BoxType "EJ3214-0000-0016"}
{attribute addProperty Id "RTD_Inputs_ChannelAT %I*ARRAY[0..6] OF RTD_Inputs_Channel_17AE08DB128160WcStateAT %I*WcState_98A4DF7520.250InfoDataAT %I*InfoData_BC63D37F80100"}
{attribute addProperty CRC "1836036553"}
{attribute addProperty SizeInBites "210"}
{attribute addProperty SizeInBytes "26.25"}
TYPE EJ3214_712ECA1B :
STRUCT
	{attribute addProperty Name "RTD_Inputs_Channel"}
	RTD_Inputs_Channel : ARRAY[0..6] OF RTD_Inputs_Channel_17AE08DB;
	{attribute addProperty Name "WcState"}
	WcState : WcState_98A4DF75;
	{attribute addProperty Name "InfoData"}
	InfoData : InfoData_BC63D37F;
END_STRUCT
END_TYPE

// ---- DUTs/IO/Boxes/EJ3255_7B3AD958.TcDUT
{attribute addProperty BoxType "EJ3255-0000-0023"}
{attribute addProperty Id "AI_Standard_ChannelAT %I*ARRAY[0..8] OF AI_Standard_Channel_087F71C7160200WcStateAT %I*WcState_98A4DF7520.250InfoDataAT %I*InfoData_BC63D37F80100"}
{attribute addProperty CRC "220768616"}
{attribute addProperty SizeInBites "242"}
{attribute addProperty SizeInBytes "30.25"}
TYPE EJ3255_7B3AD958 :
STRUCT
	{attribute addProperty Name "AI_Standard_Channel"}
	AI_Standard_Channel : ARRAY[0..8] OF AI_Standard_Channel_087F71C7;
	{attribute addProperty Name "WcState"}
	WcState : WcState_98A4DF75;
	{attribute addProperty Name "InfoData"}
	InfoData : InfoData_BC63D37F;
END_STRUCT
END_TYPE

// ---- DUTs/IO/Boxes/EJ3318_4B9E477A.TcDUT
{attribute addProperty BoxType "EJ3318-0000-0017"}
{attribute addProperty Id "TC_ChannelAT %I*ARRAY[0..14] OF TC_Channel_17AE08DB256320RTD_Inputs_ChannelAT %I*ARRAY[0..2] OF RTD_Inputs_Channel_17AE08DB6480WcStateAT %I*WcState_98A4DF7520.250InfoDataAT %I*InfoData_BC63D37F80100"}
{attribute addProperty CRC "604556167"}
{attribute addProperty SizeInBites "402"}
{attribute addProperty SizeInBytes "50.25"}
TYPE EJ3318_4B9E477A :
STRUCT
	{attribute addProperty Name "TC_Channel"}
	TC_Channel : ARRAY[0..14] OF TC_Channel_17AE08DB;
	{attribute addProperty Name "RTD_Inputs_Channel"}
	RTD_Inputs_Channel : ARRAY[0..2] OF RTD_Inputs_Channel_17AE08DB;
	{attribute addProperty Name "WcState"}
	WcState : WcState_98A4DF75;
	{attribute addProperty Name "InfoData"}
	InfoData : InfoData_BC63D37F;
END_STRUCT
END_TYPE

// ---- DUTs/IO/Boxes/EJ4002_19A75BD9.TcDUT
{attribute addProperty BoxType "EJ4002-0000-0017"}
{attribute addProperty Id "AO_Outputs_ChannelAT %Q*ARRAY[0..1] OF AO_Outputs_Channel_F57FA4F93240WcStateAT %I*WcState_28A8677510.1250InfoDataAT %I*InfoData_BC63D37F80100"}
{attribute addProperty CRC "3518482396"}
{attribute addProperty SizeInBites "113"}
{attribute addProperty SizeInBytes "14.125"}
TYPE EJ4002_19A75BD9 :
STRUCT
	{attribute addProperty Name "AO_Outputs_Channel"}
	AO_Outputs_Channel : ARRAY[0..1] OF AO_Outputs_Channel_F57FA4F9;
	{attribute addProperty Name "WcState"}
	WcState : WcState_28A86775;
	{attribute addProperty Name "InfoData"}
	InfoData : InfoData_BC63D37F;
END_STRUCT
END_TYPE

// ---- DUTs/IO/Boxes/EJ4002_BF483E01.TcDUT
{attribute addProperty BoxType "EJ4002-0000-0018"}
{attribute addProperty Id "AO_Output_ChannelAT %Q*ARRAY[0..1] OF AO_Output_Channel_F57FA4F93240WcStateAT %I*WcState_28A8677510.1250InfoDataAT %I*InfoData_BC63D37F80100"}
{attribute addProperty CRC "24542987"}
{attribute addProperty SizeInBites "113"}
{attribute addProperty SizeInBytes "14.125"}
TYPE EJ4002_BF483E01 :
STRUCT
	{attribute addProperty Name "AO_Output_Channel"}
	AO_Output_Channel : ARRAY[0..1] OF AO_Output_Channel_F57FA4F9;
	{attribute addProperty Name "WcState"}
	WcState : WcState_28A86775;
	{attribute addProperty Name "InfoData"}
	InfoData : InfoData_BC63D37F;
END_STRUCT
END_TYPE

// ---- DUTs/IO/Boxes/EJ4004_9786CACB.TcDUT
{attribute addProperty BoxType "EJ4004-0000-0020"}
{attribute addProperty Id "AO_Outputs_ChannelAT %Q*ARRAY[0..3] OF AO_Outputs_Channel_F57FA4F96480WcStateAT %I*WcState_28A8677510.1250InfoDataAT %I*InfoData_BC63D37F80100"}
{attribute addProperty CRC "854605201"}
{attribute addProperty SizeInBites "145"}
{attribute addProperty SizeInBytes "18.125"}
TYPE EJ4004_9786CACB :
STRUCT
	{attribute addProperty Name "AO_Outputs_Channel"}
	AO_Outputs_Channel : ARRAY[0..3] OF AO_Outputs_Channel_F57FA4F9;
	{attribute addProperty Name "WcState"}
	WcState : WcState_28A86775;
	{attribute addProperty Name "InfoData"}
	InfoData : InfoData_BC63D37F;
END_STRUCT
END_TYPE

// ---- DUTs/IO/Boxes/EJ4008_D5FA9EBB.TcDUT
{attribute addProperty BoxType "EJ4008-0000-0020"}
{attribute addProperty Id "AO_Outputs_ChannelAT %Q*ARRAY[0..7] OF AO_Outputs_Channel_F57FA4F9128160WcStateAT %I*WcState_28A8677510.1250InfoDataAT %I*InfoData_BC63D37F80100"}
{attribute addProperty CRC "220256351"}
{attribute addProperty SizeInBites "209"}
{attribute addProperty SizeInBytes "26.125"}
TYPE EJ4008_D5FA9EBB :
STRUCT
	{attribute addProperty Name "AO_Outputs_Channel"}
	AO_Outputs_Channel : ARRAY[0..7] OF AO_Outputs_Channel_F57FA4F9;
	{attribute addProperty Name "WcState"}
	WcState : WcState_28A86775;
	{attribute addProperty Name "InfoData"}
	InfoData : InfoData_BC63D37F;
END_STRUCT
END_TYPE

// ---- DUTs/IO/Boxes/EJ4018_D5FA9EBB.TcDUT
{attribute addProperty BoxType "EJ4018-0000-0016"}
{attribute addProperty Id "AO_Outputs_ChannelAT %Q*ARRAY[0..7] OF AO_Outputs_Channel_F57FA4F9128160WcStateAT %I*WcState_28A8677510.1250InfoDataAT %I*InfoData_BC63D37F80100"}
{attribute addProperty CRC "220256351"}
{attribute addProperty SizeInBites "209"}
{attribute addProperty SizeInBytes "26.125"}
TYPE EJ4018_D5FA9EBB :
STRUCT
	{attribute addProperty Name "AO_Outputs_Channel"}
	AO_Outputs_Channel : ARRAY[0..7] OF AO_Outputs_Channel_F57FA4F9;
	{attribute addProperty Name "WcState"}
	WcState : WcState_28A86775;
	{attribute addProperty Name "InfoData"}
	InfoData : InfoData_BC63D37F;
END_STRUCT
END_TYPE

// ---- DUTs/IO/Boxes/EJ4024_9786CACB.TcDUT
{attribute addProperty BoxType "EJ4024-0000-0020"}
{attribute addProperty Id "AO_Outputs_ChannelAT %Q*ARRAY[0..3] OF AO_Outputs_Channel_F57FA4F96480WcStateAT %I*WcState_28A8677510.1250InfoDataAT %I*InfoData_BC63D37F80100"}
{attribute addProperty CRC "854605201"}
{attribute addProperty SizeInBites "145"}
{attribute addProperty SizeInBytes "18.125"}
TYPE EJ4024_9786CACB :
STRUCT
	{attribute addProperty Name "AO_Outputs_Channel"}
	AO_Outputs_Channel : ARRAY[0..3] OF AO_Outputs_Channel_F57FA4F9;
	{attribute addProperty Name "WcState"}
	WcState : WcState_28A86775;
	{attribute addProperty Name "InfoData"}
	InfoData : InfoData_BC63D37F;
END_STRUCT
END_TYPE

// ---- DUTs/IO/Boxes/EJ4132_19A75BD9.TcDUT
{attribute addProperty BoxType "EJ4132-0000-0019"}
{attribute addProperty Id "AO_Outputs_ChannelAT %Q*ARRAY[0..1] OF AO_Outputs_Channel_F57FA4F93240WcStateAT %I*WcState_28A8677510.1250InfoDataAT %I*InfoData_BC63D37F80100"}
{attribute addProperty CRC "3518482396"}
{attribute addProperty SizeInBites "113"}
{attribute addProperty SizeInBytes "14.125"}
TYPE EJ4132_19A75BD9 :
STRUCT
	{attribute addProperty Name "AO_Outputs_Channel"}
	AO_Outputs_Channel : ARRAY[0..1] OF AO_Outputs_Channel_F57FA4F9;
	{attribute addProperty Name "WcState"}
	WcState : WcState_28A86775;
	{attribute addProperty Name "InfoData"}
	InfoData : InfoData_BC63D37F;
END_STRUCT
END_TYPE

// ---- DUTs/IO/Boxes/EJ4134_FEE36ED0.TcDUT
{attribute addProperty BoxType "EJ4134-0000-0019"}
{attribute addProperty Id "AO_Output_ChannelAT %Q*ARRAY[0..3] OF AO_Output_Channel_F57FA4F96480WcStateAT %I*WcState_28A8677510.1250InfoDataAT %I*InfoData_BC63D37F80100"}
{attribute addProperty CRC "3820990709"}
{attribute addProperty SizeInBites "145"}
{attribute addProperty SizeInBytes "18.125"}
TYPE EJ4134_FEE36ED0 :
STRUCT
	{attribute addProperty Name "AO_Output_Channel"}
	AO_Output_Channel : ARRAY[0..3] OF AO_Output_Channel_F57FA4F9;
	{attribute addProperty Name "WcState"}
	WcState : WcState_28A86775;
	{attribute addProperty Name "InfoData"}
	InfoData : InfoData_BC63D37F;
END_STRUCT
END_TYPE

// ---- DUTs/IO/Boxes/EJ5002_82283068.TcDUT
{attribute addProperty BoxType "EJ5002-0000-0016"}
{attribute addProperty Id "SSI_Inputs_ChannelAT %I*ARRAY[0..2] OF SSI_Inputs_Channel_F7D238D196120WcStateAT %I*WcState_98A4DF7520.250InfoDataAT %I*InfoData_BC63D37F80100"}
{attribute addProperty CRC "3035886411"}
{attribute addProperty SizeInBites "178"}
{attribute addProperty SizeInBytes "22.25"}
TYPE EJ5002_82283068 :
STRUCT
	{attribute addProperty Name "SSI_Inputs_Channel"}
	SSI_Inputs_Channel : ARRAY[0..2] OF SSI_Inputs_Channel_F7D238D1;
	{attribute addProperty Name "WcState"}
	WcState : WcState_98A4DF75;
	{attribute addProperty Name "InfoData"}
	InfoData : InfoData_BC63D37F;
END_STRUCT
END_TYPE

// ---- DUTs/IO/Boxes/EJ5002_960CC6F1.TcDUT
{attribute addProperty BoxType "EJ5002-0000-0017"}
{attribute addProperty Id "SSI_Inputs_ChannelAT %I*ARRAY[0..2] OF SSI_Inputs_Channel_32C7114D96120WcStateAT %I*WcState_98A4DF7520.250InfoDataAT %I*InfoData_BC63D37F80100"}
{attribute addProperty CRC "3984045230"}
{attribute addProperty SizeInBites "178"}
{attribute addProperty SizeInBytes "22.25"}
TYPE EJ5002_960CC6F1 :
STRUCT
	{attribute addProperty Name "SSI_Inputs_Channel"}
	SSI_Inputs_Channel : ARRAY[0..2] OF SSI_Inputs_Channel_32C7114D;
	{attribute addProperty Name "WcState"}
	WcState : WcState_98A4DF75;
	{attribute addProperty Name "InfoData"}
	InfoData : InfoData_BC63D37F;
END_STRUCT
END_TYPE

// ---- DUTs/IO/Boxes/EJ5101_60128726.TcDUT
{attribute addProperty BoxType "EJ5101-0000-0016"}
{attribute addProperty Id "ENC_Status_compactAT %I*ENC_Status_compact_5BAFF8F54860ENC_Control_compactAT %Q*ENC_Control_compact_03701F333240WcStateAT %I*WcState_98A4DF7520.250InfoDataAT %I*InfoData_BC63D37F80100"}
{attribute addProperty CRC "1944059784"}
{attribute addProperty SizeInBites "162"}
{attribute addProperty SizeInBytes "20.25"}
TYPE EJ5101_60128726 :
STRUCT
	{attribute addProperty Name "ENC_Status_compact"}
	ENC_Status_compact : ENC_Status_compact_5BAFF8F5;
	{attribute addProperty Name "ENC_Control_compact"}
	ENC_Control_compact : ENC_Control_compact_03701F33;
	{attribute addProperty Name "WcState"}
	WcState : WcState_98A4DF75;
	{attribute addProperty Name "InfoData"}
	InfoData : InfoData_BC63D37F;
END_STRUCT
END_TYPE

// ---- DUTs/IO/Boxes/EJ5151_0AC1A36D.TcDUT
{attribute addProperty BoxType "EJ5151-0000-0016"}
{attribute addProperty Id "ENC_InputsAT %I*ENC_Inputs_001F11BA4860ENC_Inputs_1AT %I*ENC_Inputs_AC51B8A03240ENC_OutputsAT %Q*ENC_Outputs_03701F333240WcStateAT %I*WcState_98A4DF7520.250InfoDataAT %I*InfoData_BC63D37F80100"}
{attribute addProperty CRC "2073474733"}
{attribute addProperty SizeInBites "194"}
{attribute addProperty SizeInBytes "24.25"}
TYPE EJ5151_0AC1A36D :
STRUCT
	{attribute addProperty Name "ENC_Inputs"}
	ENC_Inputs : ENC_Inputs_001F11BA;
	{attribute addProperty Name "ENC_Inputs_1"}
	ENC_Inputs_1 : ENC_Inputs_AC51B8A0;
	{attribute addProperty Name "ENC_Outputs"}
	ENC_Outputs : ENC_Outputs_03701F33;
	{attribute addProperty Name "WcState"}
	WcState : WcState_98A4DF75;
	{attribute addProperty Name "InfoData"}
	InfoData : InfoData_BC63D37F;
END_STRUCT
END_TYPE

// ---- DUTs/IO/Boxes/EJ6002_880A624E.TcDUT
{attribute addProperty BoxType "EJ6002-0000-0016"}
{attribute addProperty Id "COM_Inputs_ChannelAT %I*ARRAY[0..23] OF COM_Inputs_Channel_85D1D733384480COM_Outputs_ChannelAT %Q*ARRAY[0..23] OF COM_Outputs_Channel_85BCA431384480WcStateAT %I*WcState_98A4DF7520.250InfoDataAT %I*InfoData_BC63D37F80100"}
{attribute addProperty CRC "226543692"}
{attribute addProperty SizeInBites "850"}
{attribute addProperty SizeInBytes "106.25"}
TYPE EJ6002_880A624E :
STRUCT
	{attribute addProperty Name "COM_Inputs_Channel"}
	COM_Inputs_Channel : ARRAY[0..23] OF COM_Inputs_Channel_85D1D733;
	{attribute addProperty Name "COM_Outputs_Channel"}
	COM_Outputs_Channel : ARRAY[0..23] OF COM_Outputs_Channel_85BCA431;
	{attribute addProperty Name "WcState"}
	WcState : WcState_98A4DF75;
	{attribute addProperty Name "InfoData"}
	InfoData : InfoData_BC63D37F;
END_STRUCT
END_TYPE

// ---- DUTs/IO/Boxes/EJ6224_3990B4B4.TcDUT
{attribute addProperty BoxType "EJ6224-0000-0016"}
{attribute addProperty Id "Module_1_DeviceState_Inputs_DeviceModule_1_DeviceState_Inputs_Device_50DD3C951620Module_2_DeviceState_InputsModule_2_DeviceState_Inputs_D860B2E33240WcStateAT %I*WcState_98A4DF7520.250InfoDataAT %I*InfoData_275E3363128160"}
{attribute addProperty CRC "1978599132"}
{attribute addProperty SizeInBites "178"}
{attribute addProperty SizeInBytes "22.25"}
TYPE EJ6224_3990B4B4 :
STRUCT
	{attribute addProperty Name "Module_1_DeviceState_Inputs_Device"}
	Module_1_DeviceState_Inputs_Device : Module_1_DeviceState_Inputs_Device_50DD3C95;
	{attribute addProperty Name "Module_2_DeviceState_Inputs"}
	Module_2_DeviceState_Inputs : Module_2_DeviceState_Inputs_D860B2E3;
	{attribute addProperty Name "WcState"}
	WcState : WcState_98A4DF75;
	{attribute addProperty Name "InfoData"}
	InfoData : InfoData_275E3363;
END_STRUCT
END_TYPE

// ---- DUTs/IO/Boxes/EJ7031_26D83138.TcDUT
{attribute addProperty BoxType "EJ7031-0000-0026"}
{attribute addProperty Id "ENC_Status_compactAT %I*ENC_Status_compact_FA080ECA4860STM_StatusAT %I*STM_Status_64D937431620ENC_Control_compactAT %Q*ENC_Control_compact_5C86AA9D3240STM_ControlAT %Q*STM_Control_6F24B2C41620STM_VelocityAT %Q*STM_Velocity_1D89B5C21620WcStateAT %I*WcState_98A4DF7520.250InfoDataAT %I*InfoData_1C46E3E796120"}
{attribute addProperty CRC "1132355663"}
{attribute addProperty SizeInBites "226"}
{attribute addProperty SizeInBytes "28.25"}
TYPE EJ7031_26D83138 :
STRUCT
	{attribute addProperty Name "ENC_Status_compact"}
	ENC_Status_compact : ENC_Status_compact_FA080ECA;
	{attribute addProperty Name "STM_Status"}
	STM_Status : STM_Status_64D93743;
	{attribute addProperty Name "ENC_Control_compact"}
	ENC_Control_compact : ENC_Control_compact_5C86AA9D;
	{attribute addProperty Name "STM_Control"}
	STM_Control : STM_Control_6F24B2C4;
	{attribute addProperty Name "STM_Velocity"}
	STM_Velocity : STM_Velocity_1D89B5C2;
	{attribute addProperty Name "WcState"}
	WcState : WcState_98A4DF75;
	{attribute addProperty Name "InfoData"}
	InfoData : InfoData_1C46E3E7;
END_STRUCT
END_TYPE

// ---- DUTs/IO/Boxes/EJ7037_F30AD128.TcDUT
{attribute addProperty BoxType "EJ7037-0000-0020"}
{attribute addProperty Id "ENC_Status_compactAT %I*ENC_Status_compact_DA87336C4860STM_StatusAT %I*STM_Status_CB86BB9A1620ENC_Control_compactAT %Q*ENC_Control_compact_03701F333240STM_ControlAT %Q*STM_Control_91ECC2DE1620STM_VelocityAT %Q*STM_Velocity_1D89B5C21620WcStateAT %I*WcState_98A4DF7520.250InfoDataAT %I*InfoData_1C46E3E796120"}
{attribute addProperty CRC "1249776780"}
{attribute addProperty SizeInBites "226"}
{attribute addProperty SizeInBytes "28.25"}
TYPE EJ7037_F30AD128 :
STRUCT
	{attribute addProperty Name "ENC_Status_compact"}
	ENC_Status_compact : ENC_Status_compact_DA87336C;
	{attribute addProperty Name "STM_Status"}
	STM_Status : STM_Status_CB86BB9A;
	{attribute addProperty Name "ENC_Control_compact"}
	ENC_Control_compact : ENC_Control_compact_03701F33;
	{attribute addProperty Name "STM_Control"}
	STM_Control : STM_Control_91ECC2DE;
	{attribute addProperty Name "STM_Velocity"}
	STM_Velocity : STM_Velocity_1D89B5C2;
	{attribute addProperty Name "WcState"}
	WcState : WcState_98A4DF75;
	{attribute addProperty Name "InfoData"}
	InfoData : InfoData_1C46E3E7;
END_STRUCT
END_TYPE

// ---- DUTs/IO/Boxes/EJ7041_26D83138.TcDUT
{attribute addProperty BoxType "EJ7041-0052-0016"}
{attribute addProperty Id "ENC_Status_compactAT %I*ENC_Status_compact_FA080ECA4860STM_StatusAT %I*STM_Status_64D937431620ENC_Control_compactAT %Q*ENC_Control_compact_5C86AA9D3240STM_ControlAT %Q*STM_Control_6F24B2C41620STM_VelocityAT %Q*STM_Velocity_1D89B5C21620WcStateAT %I*WcState_98A4DF7520.250InfoDataAT %I*InfoData_1C46E3E796120"}
{attribute addProperty CRC "1132355663"}
{attribute addProperty SizeInBites "226"}
{attribute addProperty SizeInBytes "28.25"}
TYPE EJ7041_26D83138 :
STRUCT
	{attribute addProperty Name "ENC_Status_compact"}
	ENC_Status_compact : ENC_Status_compact_FA080ECA;
	{attribute addProperty Name "STM_Status"}
	STM_Status : STM_Status_64D93743;
	{attribute addProperty Name "ENC_Control_compact"}
	ENC_Control_compact : ENC_Control_compact_5C86AA9D;
	{attribute addProperty Name "STM_Control"}
	STM_Control : STM_Control_6F24B2C4;
	{attribute addProperty Name "STM_Velocity"}
	STM_Velocity : STM_Velocity_1D89B5C2;
	{attribute addProperty Name "WcState"}
	WcState : WcState_98A4DF75;
	{attribute addProperty Name "InfoData"}
	InfoData : InfoData_1C46E3E7;
END_STRUCT
END_TYPE

// ---- DUTs/IO/Boxes/EJ7047_F30AD128.TcDUT
{attribute addProperty BoxType "EJ7047-0000-0018"}
{attribute addProperty Id "ENC_Status_compactAT %I*ENC_Status_compact_DA87336C4860STM_StatusAT %I*STM_Status_CB86BB9A1620ENC_Control_compactAT %Q*ENC_Control_compact_03701F333240STM_ControlAT %Q*STM_Control_91ECC2DE1620STM_VelocityAT %Q*STM_Velocity_1D89B5C21620WcStateAT %I*WcState_98A4DF7520.250InfoDataAT %I*InfoData_1C46E3E796120"}
{attribute addProperty CRC "1249776780"}
{attribute addProperty SizeInBites "226"}
{attribute addProperty SizeInBytes "28.25"}
TYPE EJ7047_F30AD128 :
STRUCT
	{attribute addProperty Name "ENC_Status_compact"}
	ENC_Status_compact : ENC_Status_compact_DA87336C;
	{attribute addProperty Name "STM_Status"}
	STM_Status : STM_Status_CB86BB9A;
	{attribute addProperty Name "ENC_Control_compact"}
	ENC_Control_compact : ENC_Control_compact_03701F33;
	{attribute addProperty Name "STM_Control"}
	STM_Control : STM_Control_91ECC2DE;
	{attribute addProperty Name "STM_Velocity"}
	STM_Velocity : STM_Velocity_1D89B5C2;
	{attribute addProperty Name "WcState"}
	WcState : WcState_98A4DF75;
	{attribute addProperty Name "InfoData"}
	InfoData : InfoData_1C46E3E7;
END_STRUCT
END_TYPE

// ---- DUTs/IO/Boxes/EJ7342_E03DC371.TcDUT
{attribute addProperty BoxType "EJ7342-0000-0019"}
{attribute addProperty Id "ENC_Status_compact_ChannelAT %I*ARRAY[0..3] OF ENC_Status_compact_Channel_559DED9896120DCM_Status_ChannelAT %I*ARRAY[0..1] OF DCM_Status_Channel_C2B0CAE13240ENC_Control_compact_ChannelAT %Q*ARRAY[0..2] OF ENC_Control_compact_Channel_5C86AA9D6480DCM_Control_Channel_1AT %Q*DCM_Control_Channel_6F24B2C41620DCM_Velocity_Channel_1AT %Q*DCM_Velocity_Channel_1D89B5C21620DCM_Control_Channel_2AT %Q*DCM_Control_Channel_6F24B2C41620DCM_Velocity_Channel_2AT %Q*DCM_Velocity_Channel_1D89B5C21620WcStateAT %I*WcState_98A4DF7520.250InfoDataAT %I*InfoData_3F3BB279112140"}
{attribute addProperty CRC "69007491"}
{attribute addProperty SizeInBites "370"}
{attribute addProperty SizeInBytes "46.25"}
TYPE EJ7342_E03DC371 :
STRUCT
	{attribute addProperty Name "ENC_Status_compact_Channel"}
	ENC_Status_compact_Channel : ARRAY[0..3] OF ENC_Status_compact_Channel_559DED98;
	{attribute addProperty Name "DCM_Status_Channel"}
	DCM_Status_Channel : ARRAY[0..1] OF DCM_Status_Channel_C2B0CAE1;
	{attribute addProperty Name "ENC_Control_compact_Channel"}
	ENC_Control_compact_Channel : ARRAY[0..2] OF ENC_Control_compact_Channel_5C86AA9D;
	{attribute addProperty Name "DCM_Control_Channel_1"}
	DCM_Control_Channel_1 : DCM_Control_Channel_6F24B2C4;
	{attribute addProperty Name "DCM_Velocity_Channel_1"}
	DCM_Velocity_Channel_1 : DCM_Velocity_Channel_1D89B5C2;
	{attribute addProperty Name "DCM_Control_Channel_2"}
	DCM_Control_Channel_2 : DCM_Control_Channel_6F24B2C4;
	{attribute addProperty Name "DCM_Velocity_Channel_2"}
	DCM_Velocity_Channel_2 : DCM_Velocity_Channel_1D89B5C2;
	{attribute addProperty Name "WcState"}
	WcState : WcState_98A4DF75;
	{attribute addProperty Name "InfoData"}
	InfoData : InfoData_3F3BB279;
END_STRUCT
END_TYPE

// ---- DUTs/IO/Boxes/EJ7342_E2585B83.TcDUT
{attribute addProperty BoxType "EJ7342-0000-0020"}
{attribute addProperty Id "ENC_Status_compact_ChannelAT %I*ARRAY[0..3] OF ENC_Status_compact_Channel_A7E8355C96120DCM_Status_ChannelAT %I*ARRAY[0..1] OF DCM_Status_Channel_64D937433240ENC_Control_compact_ChannelAT %Q*ARRAY[0..2] OF ENC_Control_compact_Channel_5C86AA9D6480DCM_Control_Channel_1AT %Q*DCM_Control_Channel_6F24B2C41620DCM_Velocity_Channel_1AT %Q*DCM_Velocity_Channel_1D89B5C21620DCM_Control_Channel_2AT %Q*DCM_Control_Channel_6F24B2C41620DCM_Velocity_Channel_2AT %Q*DCM_Velocity_Channel_1D89B5C21620WcStateAT %I*WcState_98A4DF7520.250InfoDataAT %I*InfoData_3F3BB279112140"}
{attribute addProperty CRC "3764429889"}
{attribute addProperty SizeInBites "370"}
{attribute addProperty SizeInBytes "46.25"}
TYPE EJ7342_E2585B83 :
STRUCT
	{attribute addProperty Name "ENC_Status_compact_Channel"}
	ENC_Status_compact_Channel : ARRAY[0..3] OF ENC_Status_compact_Channel_A7E8355C;
	{attribute addProperty Name "DCM_Status_Channel"}
	DCM_Status_Channel : ARRAY[0..1] OF DCM_Status_Channel_64D93743;
	{attribute addProperty Name "ENC_Control_compact_Channel"}
	ENC_Control_compact_Channel : ARRAY[0..2] OF ENC_Control_compact_Channel_5C86AA9D;
	{attribute addProperty Name "DCM_Control_Channel_1"}
	DCM_Control_Channel_1 : DCM_Control_Channel_6F24B2C4;
	{attribute addProperty Name "DCM_Velocity_Channel_1"}
	DCM_Velocity_Channel_1 : DCM_Velocity_Channel_1D89B5C2;
	{attribute addProperty Name "DCM_Control_Channel_2"}
	DCM_Control_Channel_2 : DCM_Control_Channel_6F24B2C4;
	{attribute addProperty Name "DCM_Velocity_Channel_2"}
	DCM_Velocity_Channel_2 : DCM_Velocity_Channel_1D89B5C2;
	{attribute addProperty Name "WcState"}
	WcState : WcState_98A4DF75;
	{attribute addProperty Name "InfoData"}
	InfoData : InfoData_3F3BB279;
END_STRUCT
END_TYPE

// ---- DUTs/IO/Boxes/EJ7211_83D4128E.TcDUT
{attribute addProperty BoxType "EJ7211-0010-0026"}
{attribute addProperty Id "FB_PositionAT %I*FB_Position_BA8AA9F03240DRV_StatuswordAT %I*DRV_Statusword_53CBCECC1620DRV_ControlwordAT %Q*DRV_Controlword_417617681620DRV_Target_velocityAT %Q*DRV_Target_velocity_53A88AB03240WcStateAT %I*WcState_98A4DF7520.250InfoDataAT %I*InfoData_AEB17F4D152190"}
{attribute addProperty CRC "777447930"}
{attribute addProperty SizeInBites "250"}
{attribute addProperty SizeInBytes "31.25"}
TYPE EJ7211_83D4128E :
STRUCT
	{attribute addProperty Name "FB_Position"}
	FB_Position : FB_Position_BA8AA9F0;
	{attribute addProperty Name "DRV_Statusword"}
	DRV_Statusword : DRV_Statusword_53CBCECC;
	{attribute addProperty Name "DRV_Controlword"}
	DRV_Controlword : DRV_Controlword_41761768;
	{attribute addProperty Name "DRV_Target_velocity"}
	DRV_Target_velocity : DRV_Target_velocity_53A88AB0;
	{attribute addProperty Name "WcState"}
	WcState : WcState_98A4DF75;
	{attribute addProperty Name "InfoData"}
	InfoData : InfoData_AEB17F4D;
END_STRUCT
END_TYPE

// ---- DUTs/IO/Boxes/EJ7211_2D7B43DC.TcDUT
{attribute addProperty BoxType "EJ7211-0010-0030"}
{attribute addProperty Id "FB_PositionAT %I*FB_Position_BA8AA9F03240DRV_StatuswordAT %I*DRV_Statusword_53CBCECC1620DRV_ControlwordAT %Q*DRV_Controlword_417617681620DRV_Target_velocityAT %Q*DRV_Target_velocity_53A88AB03240WcStateAT %I*WcState_98A4DF7520.250InfoDataAT %I*InfoData_81099714160200"}
{attribute addProperty CRC "1285967358"}
{attribute addProperty SizeInBites "258"}
{attribute addProperty SizeInBytes "32.25"}
TYPE EJ7211_2D7B43DC :
STRUCT
	{attribute addProperty Name "FB_Position"}
	FB_Position : FB_Position_BA8AA9F0;
	{attribute addProperty Name "DRV_Statusword"}
	DRV_Statusword : DRV_Statusword_53CBCECC;
	{attribute addProperty Name "DRV_Controlword"}
	DRV_Controlword : DRV_Controlword_41761768;
	{attribute addProperty Name "DRV_Target_velocity"}
	DRV_Target_velocity : DRV_Target_velocity_53A88AB0;
	{attribute addProperty Name "WcState"}
	WcState : WcState_98A4DF75;
	{attribute addProperty Name "InfoData"}
	InfoData : InfoData_81099714;
END_STRUCT
END_TYPE

// ---- DUTs/IO/Boxes/EJ7211_789C0F59.TcDUT
{attribute addProperty BoxType "EJ7211-0011-0026"}
{attribute addProperty Id "DS402_StatuswordAT %I*DS402_Statusword_53CBCECC1620DS402_Position_actual_valueAT %I*DS402_Position_actual_value_0D11C1143240DS402_ControlwordAT %Q*DS402_Controlword_417617681620DS402_Target_velocityAT %Q*DS402_Target_velocity_53A88AB03240WcStateAT %I*WcState_98A4DF7520.250InfoDataAT %I*InfoData_AEB17F4D152190"}
{attribute addProperty CRC "2160702565"}
{attribute addProperty SizeInBites "250"}
{attribute addProperty SizeInBytes "31.25"}
TYPE EJ7211_789C0F59 :
STRUCT
	{attribute addProperty Name "DS402_Statusword"}
	DS402_Statusword : DS402_Statusword_53CBCECC;
	{attribute addProperty Name "DS402_Position_actual_value"}
	DS402_Position_actual_value : DS402_Position_actual_value_0D11C114;
	{attribute addProperty Name "DS402_Controlword"}
	DS402_Controlword : DS402_Controlword_41761768;
	{attribute addProperty Name "DS402_Target_velocity"}
	DS402_Target_velocity : DS402_Target_velocity_53A88AB0;
	{attribute addProperty Name "WcState"}
	WcState : WcState_98A4DF75;
	{attribute addProperty Name "InfoData"}
	InfoData : InfoData_AEB17F4D;
END_STRUCT
END_TYPE

// ---- DUTs/IO/Boxes/EJ7211_5D870918.TcDUT
{attribute addProperty BoxType "EJ7211-9414-0030"}
{attribute addProperty Id "FB_PositionAT %I*FB_Position_BA8AA9F03240DRV_StatuswordAT %I*DRV_Statusword_53CBCECC1620DRV_ControlwordAT %Q*DRV_Controlword_417617681620DRV_Target_velocityAT %Q*DRV_Target_velocity_53A88AB03240WcStateAT %I*WcState_98A4DF7520.250InfoDataAT %I*InfoData_BF6E01EA168210"}
{attribute addProperty CRC "1347982361"}
{attribute addProperty SizeInBites "266"}
{attribute addProperty SizeInBytes "33.25"}
TYPE EJ7211_5D870918 :
STRUCT
	{attribute addProperty Name "FB_Position"}
	FB_Position : FB_Position_BA8AA9F0;
	{attribute addProperty Name "DRV_Statusword"}
	DRV_Statusword : DRV_Statusword_53CBCECC;
	{attribute addProperty Name "DRV_Controlword"}
	DRV_Controlword : DRV_Controlword_41761768;
	{attribute addProperty Name "DRV_Target_velocity"}
	DRV_Target_velocity : DRV_Target_velocity_53A88AB0;
	{attribute addProperty Name "WcState"}
	WcState : WcState_98A4DF75;
	{attribute addProperty Name "InfoData"}
	InfoData : InfoData_BF6E01EA;
END_STRUCT
END_TYPE

// ---- DUTs/IO/Boxes/EJ7334_68079CA9.TcDUT
{attribute addProperty BoxType "EJ7334-0008-0016"}
{attribute addProperty Id "DCM_Status_ChannelAT %I*ARRAY[0..3] OF DCM_Status_Channel_DBE0EA1F6480DCM_Outputs_ChannelAT %Q*ARRAY[0..6] OF DCM_Outputs_Channel_1F77C8C2128160WcStateAT %I*WcState_98A4DF7520.250InfoDataAT %I*InfoData_BC63D37F80100"}
{attribute addProperty CRC "3805991956"}
{attribute addProperty SizeInBites "274"}
{attribute addProperty SizeInBytes "34.25"}
TYPE EJ7334_68079CA9 :
STRUCT
	{attribute addProperty Name "DCM_Status_Channel"}
	DCM_Status_Channel : ARRAY[0..3] OF DCM_Status_Channel_DBE0EA1F;
	{attribute addProperty Name "DCM_Outputs_Channel"}
	DCM_Outputs_Channel : ARRAY[0..6] OF DCM_Outputs_Channel_1F77C8C2;
	{attribute addProperty Name "WcState"}
	WcState : WcState_98A4DF75;
	{attribute addProperty Name "InfoData"}
	InfoData : InfoData_BC63D37F;
END_STRUCT
END_TYPE

// ---- DUTs/IO/Boxes/EJ7411_675FBD05.TcDUT
{attribute addProperty BoxType "EJ7411-0000-0018"}
{attribute addProperty Id "FB_PositionAT %I*FB_Position_BA8AA9F03240DRV_StatuswordAT %I*DRV_Statusword_53CBCECC1620DRV_Following_error_actual_valueAT %I*DRV_Following_error_actual_value_F54335363240DRV_ControlwordAT %Q*DRV_Controlword_417617681620DRV_Target_positionAT %Q*DRV_Target_position_41334FAA3240WcStateAT %I*WcState_98A4DF7520.250InfoDataAT %I*InfoData_81099714160200"}
{attribute addProperty CRC "4078408466"}
{attribute addProperty SizeInBites "290"}
{attribute addProperty SizeInBytes "36.25"}
TYPE EJ7411_675FBD05 :
STRUCT
	{attribute addProperty Name "FB_Position"}
	FB_Position : FB_Position_BA8AA9F0;
	{attribute addProperty Name "DRV_Statusword"}
	DRV_Statusword : DRV_Statusword_53CBCECC;
	{attribute addProperty Name "DRV_Following_error_actual_value"}
	DRV_Following_error_actual_value : DRV_Following_error_actual_value_F5433536;
	{attribute addProperty Name "DRV_Controlword"}
	DRV_Controlword : DRV_Controlword_41761768;
	{attribute addProperty Name "DRV_Target_position"}
	DRV_Target_position : DRV_Target_position_41334FAA;
	{attribute addProperty Name "WcState"}
	WcState : WcState_98A4DF75;
	{attribute addProperty Name "InfoData"}
	InfoData : InfoData_81099714;
END_STRUCT
END_TYPE

// ---- DUTs/IO/Boxes/EJ9001_179A0949.TcDUT
{attribute addProperty BoxType "EJ9001-0000-0016"}
{attribute addProperty Id "InfoDataInfoData_192954DE162"}
{attribute addProperty CRC "395970889"}
{attribute addProperty SizeInBites "16"}
{attribute addProperty SizeInBytes "2"}
TYPE EJ9001_179A0949 :
STRUCT
	{attribute addProperty Name "InfoData"}
	InfoData : InfoData_192954DE;
END_STRUCT
END_TYPE

// ---- DUTs/IO/Boxes/EJ9505_13AAEB7E.TcDUT
{attribute addProperty BoxType "EJ9505-0000-0016"}
{attribute addProperty Id "Status_UoAT %I*Status_Uo_D24303661620WcStateAT %I*WcState_98A4DF7520.250InfoDataAT %I*InfoData_192954DE1620"}
{attribute addProperty CRC "1126846400"}
{attribute addProperty SizeInBites "34"}
{attribute addProperty SizeInBytes "4.25"}
TYPE EJ9505_13AAEB7E :
STRUCT
	{attribute addProperty Name "Status_Uo"}
	Status_Uo : Status_Uo_D2430366;
	{attribute addProperty Name "WcState"}
	WcState : WcState_98A4DF75;
	{attribute addProperty Name "InfoData"}
	InfoData : InfoData_192954DE;
END_STRUCT
END_TYPE

// ---- DUTs/IO/Boxes/EJ9576_30D5723B.TcDUT
{attribute addProperty BoxType "EJ9576-0000-0018"}
{attribute addProperty Id "BCT_InputsAT %I*BCT_Inputs_7F924099128160WcStateAT %I*WcState_98A4DF7520.250InfoDataAT %I*InfoData_BC63D37F80100"}
{attribute addProperty CRC "3669577925"}
{attribute addProperty SizeInBites "210"}
{attribute addProperty SizeInBytes "26.25"}
TYPE EJ9576_30D5723B :
STRUCT
	{attribute addProperty Name "BCT_Inputs"}
	BCT_Inputs : BCT_Inputs_7F924099;
	{attribute addProperty Name "WcState"}
	WcState : WcState_98A4DF75;
	{attribute addProperty Name "InfoData"}
	InfoData : InfoData_BC63D37F;
END_STRUCT
END_TYPE

// ---- DUTs/IO/Boxes/EJ9576_8602C5C4.TcDUT
{attribute addProperty BoxType "EJ9576-0000-0019"}
{attribute addProperty Id "BCT_InputsAT %I*BCT_Inputs_6A3D8194136170WcStateAT %I*WcState_98A4DF7520.250InfoDataAT %I*InfoData_BC63D37F80100"}
{attribute addProperty CRC "66584641"}
{attribute addProperty SizeInBites "218"}
{attribute addProperty SizeInBytes "27.25"}
TYPE EJ9576_8602C5C4 :
STRUCT
	{attribute addProperty Name "BCT_Inputs"}
	BCT_Inputs : BCT_Inputs_6A3D8194;
	{attribute addProperty Name "WcState"}
	WcState : WcState_98A4DF75;
	{attribute addProperty Name "InfoData"}
	InfoData : InfoData_BC63D37F;
END_STRUCT
END_TYPE

// ---- DUTs/IO/Boxes/EJ9576_EB67CEB4.TcDUT
{attribute addProperty BoxType "EJ9576-0000-0020"}
{attribute addProperty Id "BCT_InputsAT %I*BCT_Inputs_047F8208128160WcStateAT %I*WcState_98A4DF7520.250InfoDataAT %I*InfoData_BC63D37F80100"}
{attribute addProperty CRC "903969579"}
{attribute addProperty SizeInBites "210"}
{attribute addProperty SizeInBytes "26.25"}
TYPE EJ9576_EB67CEB4 :
STRUCT
	{attribute addProperty Name "BCT_Inputs"}
	BCT_Inputs : BCT_Inputs_047F8208;
	{attribute addProperty Name "WcState"}
	WcState : WcState_98A4DF75;
	{attribute addProperty Name "InfoData"}
	InfoData : InfoData_BC63D37F;
END_STRUCT
END_TYPE

// ---- DUTs/IO/Boxes/EJ9576_EEF16252.TcDUT
{attribute addProperty BoxType "EJ9576-0000-0022"}
{attribute addProperty Id "BCT_InputsAT %I*BCT_Inputs_4FFA390D136170WcStateAT %I*WcState_98A4DF7520.250InfoDataAT %I*InfoData_BC63D37F80100"}
{attribute addProperty CRC "3662139758"}
{attribute addProperty SizeInBites "218"}
{attribute addProperty SizeInBytes "27.25"}
TYPE EJ9576_EEF16252 :
STRUCT
	{attribute addProperty Name "BCT_Inputs"}
	BCT_Inputs : BCT_Inputs_4FFA390D;
	{attribute addProperty Name "WcState"}
	WcState : WcState_98A4DF75;
	{attribute addProperty Name "InfoData"}
	InfoData : InfoData_BC63D37F;
END_STRUCT
END_TYPE

// ---- DUTs/IO/Boxes/EJ1914_5EB96E2D.TcDUT
{attribute addProperty BoxType "EJ1914-0000-0017"}
{attribute addProperty Id "Module_1_FSOEModule_1_FSOE_6091994196120Module_2_DEVICEIOModule_2_DEVICEIO_FB2B67D71620Module_3_FSLOGICModule_3_FSLOGIC_3E6251391620WcStateAT %I*WcState_98A4DF7520.250InfoDataAT %I*InfoData_BC63D37F80100"}
{attribute addProperty CRC "462638421"}
{attribute addProperty SizeInBites "210"}
{attribute addProperty SizeInBytes "26.25"}
TYPE EJ1914_5EB96E2D :
STRUCT
	{attribute addProperty Name "Module_1_FSOE"}
	Module_1_FSOE : Module_1_FSOE_60919941;
	{attribute addProperty Name "Module_2_DEVICEIO"}
	Module_2_DEVICEIO : Module_2_DEVICEIO_FB2B67D7;
	{attribute addProperty Name "Module_3_FSLOGIC"}
	Module_3_FSLOGIC : Module_3_FSLOGIC_3E625139;
	{attribute addProperty Name "WcState"}
	WcState : WcState_98A4DF75;
	{attribute addProperty Name "InfoData"}
	InfoData : InfoData_BC63D37F;
END_STRUCT
END_TYPE

// ---- DUTs/IO/Boxes/EJ1918_151E5A82.TcDUT
{attribute addProperty BoxType "EJ1918-0000-0017"}
{attribute addProperty Id "Module_1_FSOEModule_1_FSOE_99CFC0AE104130Module_2_DEVICEIOModule_2_DEVICEIO_FB2B67D71620Module_3_FSLOGICModule_3_FSLOGIC_3E6251391620WcStateAT %I*WcState_98A4DF7520.250InfoDataAT %I*InfoData_BC63D37F80100"}
{attribute addProperty CRC "3580821133"}
{attribute addProperty SizeInBites "218"}
{attribute addProperty SizeInBytes "27.25"}
TYPE EJ1918_151E5A82 :
STRUCT
	{attribute addProperty Name "Module_1_FSOE"}
	Module_1_FSOE : Module_1_FSOE_99CFC0AE;
	{attribute addProperty Name "Module_2_DEVICEIO"}
	Module_2_DEVICEIO : Module_2_DEVICEIO_FB2B67D7;
	{attribute addProperty Name "Module_3_FSLOGIC"}
	Module_3_FSLOGIC : Module_3_FSLOGIC_3E625139;
	{attribute addProperty Name "WcState"}
	WcState : WcState_98A4DF75;
	{attribute addProperty Name "InfoData"}
	InfoData : InfoData_BC63D37F;
END_STRUCT
END_TYPE

// ---- DUTs/IO/Boxes/EJ1957_6B6926D1.TcDUT
{attribute addProperty BoxType "EJ1957-0000-0017"}
{attribute addProperty Id "Module_1_FSOEModule_1_FSOE_B52BB714112140Module_2_FSOUTModule_2_FSOUT_B889B7D03240Module_3_DEVICEIOModule_3_DEVICEIO_FB2B67D71620Module_4_FSLOGICModule_4_FSLOGIC_3E6251391620WcStateAT %I*WcState_DC9C971540.50InfoDataAT %I*InfoData_BC63D37F80100"}
{attribute addProperty CRC "2859848888"}
{attribute addProperty SizeInBites "260"}
{attribute addProperty SizeInBytes "32.5"}
TYPE EJ1957_6B6926D1 :
STRUCT
	{attribute addProperty Name "Module_1_FSOE"}
	Module_1_FSOE : Module_1_FSOE_B52BB714;
	{attribute addProperty Name "Module_2_FSOUT"}
	Module_2_FSOUT : Module_2_FSOUT_B889B7D0;
	{attribute addProperty Name "Module_3_DEVICEIO"}
	Module_3_DEVICEIO : Module_3_DEVICEIO_FB2B67D7;
	{attribute addProperty Name "Module_4_FSLOGIC"}
	Module_4_FSLOGIC : Module_4_FSLOGIC_3E625139;
	{attribute addProperty Name "WcState"}
	WcState : WcState_DC9C9715;
	{attribute addProperty Name "InfoData"}
	InfoData : InfoData_BC63D37F;
END_STRUCT
END_TYPE

// ---- DUTs/IO/Boxes/EJ2914_46D107EB.TcDUT
{attribute addProperty BoxType "EJ2914-0000-0017"}
{attribute addProperty Id "Module_1_FSOEModule_1_FSOE_D19648F396120Module_2_FSOUTModule_2_FSOUT_B889B7D03240Module_3_DEVICEIOModule_3_DEVICEIO_FB2B67D71620Module_4_FSLOGICModule_4_FSLOGIC_3E6251391620WcStateAT %I*WcState_DC9C971540.50InfoDataAT %I*InfoData_BC63D37F80100"}
{attribute addProperty CRC "213205681"}
{attribute addProperty SizeInBites "244"}
{attribute addProperty SizeInBytes "30.5"}
TYPE EJ2914_46D107EB :
STRUCT
	{attribute addProperty Name "Module_1_FSOE"}
	Module_1_FSOE : Module_1_FSOE_D19648F3;
	{attribute addProperty Name "Module_2_FSOUT"}
	Module_2_FSOUT : Module_2_FSOUT_B889B7D0;
	{attribute addProperty Name "Module_3_DEVICEIO"}
	Module_3_DEVICEIO : Module_3_DEVICEIO_FB2B67D7;
	{attribute addProperty Name "Module_4_FSLOGIC"}
	Module_4_FSLOGIC : Module_4_FSLOGIC_3E625139;
	{attribute addProperty Name "WcState"}
	WcState : WcState_DC9C9715;
	{attribute addProperty Name "InfoData"}
	InfoData : InfoData_BC63D37F;
END_STRUCT
END_TYPE

// ---- DUTs/IO/Boxes/EJ2918_AA36864B.TcDUT
{attribute addProperty BoxType "EJ2918-0000-0017"}
{attribute addProperty Id "Module_1_FSOEModule_1_FSOE_FC73D945104130Module_2_FSOUTModule_2_FSOUT_15E085466480Module_3_DEVICEIOModule_3_DEVICEIO_FB2B67D71620Module_4_FSLOGICModule_4_FSLOGIC_3E6251391620WcStateAT %I*WcState_DC9C971540.50InfoDataAT %I*InfoData_BC63D37F80100"}
{attribute addProperty CRC "2831312890"}
{attribute addProperty SizeInBites "284"}
{attribute addProperty SizeInBytes "35.5"}
TYPE EJ2918_AA36864B :
STRUCT
	{attribute addProperty Name "Module_1_FSOE"}
	Module_1_FSOE : Module_1_FSOE_FC73D945;
	{attribute addProperty Name "Module_2_FSOUT"}
	Module_2_FSOUT : Module_2_FSOUT_15E08546;
	{attribute addProperty Name "Module_3_DEVICEIO"}
	Module_3_DEVICEIO : Module_3_DEVICEIO_FB2B67D7;
	{attribute addProperty Name "Module_4_FSLOGIC"}
	Module_4_FSLOGIC : Module_4_FSLOGIC_3E625139;
	{attribute addProperty Name "WcState"}
	WcState : WcState_DC9C9715;
	{attribute addProperty Name "InfoData"}
	InfoData : InfoData_BC63D37F;
END_STRUCT
END_TYPE

// ---- DUTs/IO/Boxes/EJ6910_4EA245C6.TcDUT
{attribute addProperty BoxType "EJ6910-0000-0018"}
{attribute addProperty Id "FSLOGIC_InputsAT %I*FSLOGIC_Inputs_8BA5C9331620FSLOGIC_OutputsAT %Q*EMPTY_STRUCTURE000WcStateAT %I*WcState_98A4DF7520.250InfoDataAT %I*InfoData_BC63D37F80100"}
{attribute addProperty CRC "1002942579"}
{attribute addProperty SizeInBites "98"}
{attribute addProperty SizeInBytes "12.25"}
TYPE EJ6910_4EA245C6 :
STRUCT
	{attribute addProperty Name "FSLOGIC_Inputs"}
	FSLOGIC_Inputs : FSLOGIC_Inputs_8BA5C933;
	{attribute addProperty Name "FSLOGIC_Outputs"}
	FSLOGIC_Outputs : EMPTY_STRUCTURE;
	{attribute addProperty Name "WcState"}
	WcState : WcState_98A4DF75;
	{attribute addProperty Name "InfoData"}
	InfoData : InfoData_BC63D37F;
END_STRUCT
END_TYPE

// ---- DUTs/IO/Boxes/EK1101_963BF4D7.TcDUT
{attribute addProperty BoxType "EK1101-0000-0016"}
{attribute addProperty Id "IDAT %I*ID_90FEAF081620WcStateAT %I*WcState_98A4DF7520.250InfoDataAT %I*InfoData_192954DE1620"}
{attribute addProperty CRC "1114059904"}
{attribute addProperty SizeInBites "34"}
{attribute addProperty SizeInBytes "4.25"}
TYPE EK1101_963BF4D7 :
STRUCT
	{attribute addProperty Name "ID"}
	ID : ID_90FEAF08;
	{attribute addProperty Name "WcState"}
	WcState : WcState_98A4DF75;
	{attribute addProperty Name "InfoData"}
	InfoData : InfoData_192954DE;
END_STRUCT
END_TYPE

// ---- DUTs/IO/Boxes/EK1110_179A0949.TcDUT
{attribute addProperty BoxType "EK1110-0043-0016"}
{attribute addProperty Id "InfoDataInfoData_192954DE162"}
{attribute addProperty CRC "395970889"}
{attribute addProperty SizeInBites "16"}
{attribute addProperty SizeInBytes "2"}
TYPE EK1110_179A0949 :
STRUCT
	{attribute addProperty Name "InfoData"}
	InfoData : InfoData_192954DE;
END_STRUCT
END_TYPE

// ---- DUTs/IO/Boxes/EK1121_179A0949.TcDUT
{attribute addProperty BoxType "EK1121-0010-0016"}
{attribute addProperty Id "InfoDataInfoData_192954DE162"}
{attribute addProperty CRC "395970889"}
{attribute addProperty SizeInBites "16"}
{attribute addProperty SizeInBytes "2"}
TYPE EK1121_179A0949 :
STRUCT
	{attribute addProperty Name "InfoData"}
	InfoData : InfoData_192954DE;
END_STRUCT
END_TYPE

// ---- DUTs/IO/Boxes/EK1300_0EEAC8F2.TcDUT
{attribute addProperty BoxType "EK1300-0000-0017"}
{attribute addProperty Id "Status_UsAT %I*Status_Us_D944C060810Status_UpAT %I*Status_Up_D944C060810WcStateAT %I*WcState_98A4DF7520.250InfoDataAT %I*InfoData_192954DE1620"}
{attribute addProperty CRC "793642750"}
{attribute addProperty SizeInBites "34"}
{attribute addProperty SizeInBytes "4.25"}
TYPE EK1300_0EEAC8F2 :
STRUCT
	{attribute addProperty Name "Status_Us"}
	Status_Us : Status_Us_D944C060;
	{attribute addProperty Name "Status_Up"}
	Status_Up : Status_Up_D944C060;
	{attribute addProperty Name "WcState"}
	WcState : WcState_98A4DF75;
	{attribute addProperty Name "InfoData"}
	InfoData : InfoData_192954DE;
END_STRUCT
END_TYPE

// ---- DUTs/IO/Boxes/EK1322_0EEAC8F2.TcDUT
{attribute addProperty BoxType "EK1322-0000-0017"}
{attribute addProperty Id "Status_UsAT %I*Status_Us_D944C060810Status_UpAT %I*Status_Up_D944C060810WcStateAT %I*WcState_98A4DF7520.250InfoDataAT %I*InfoData_192954DE1620"}
{attribute addProperty CRC "793642750"}
{attribute addProperty SizeInBites "34"}
{attribute addProperty SizeInBytes "4.25"}
TYPE EK1322_0EEAC8F2 :
STRUCT
	{attribute addProperty Name "Status_Us"}
	Status_Us : Status_Us_D944C060;
	{attribute addProperty Name "Status_Up"}
	Status_Up : Status_Up_D944C060;
	{attribute addProperty Name "WcState"}
	WcState : WcState_98A4DF75;
	{attribute addProperty Name "InfoData"}
	InfoData : InfoData_192954DE;
END_STRUCT
END_TYPE

// ---- DUTs/IO/Boxes/EK1310_0EEAC8F2.TcDUT
{attribute addProperty BoxType "EK1310-0000-0017"}
{attribute addProperty Id "Status_UsAT %I*Status_Us_D944C060810Status_UpAT %I*Status_Up_D944C060810WcStateAT %I*WcState_98A4DF7520.250InfoDataAT %I*InfoData_192954DE1620"}
{attribute addProperty CRC "793642750"}
{attribute addProperty SizeInBites "34"}
{attribute addProperty SizeInBytes "4.25"}
TYPE EK1310_0EEAC8F2 :
STRUCT
	{attribute addProperty Name "Status_Us"}
	Status_Us : Status_Us_D944C060;
	{attribute addProperty Name "Status_Up"}
	Status_Up : Status_Up_D944C060;
	{attribute addProperty Name "WcState"}
	WcState : WcState_98A4DF75;
	{attribute addProperty Name "InfoData"}
	InfoData : InfoData_192954DE;
END_STRUCT
END_TYPE

// ---- DUTs/IO/Boxes/EK1501_963BF4D7.TcDUT
{attribute addProperty BoxType "EK1501-0000-0016"}
{attribute addProperty Id "IDAT %I*ID_90FEAF081620WcStateAT %I*WcState_98A4DF7520.250InfoDataAT %I*InfoData_192954DE1620"}
{attribute addProperty CRC "1114059904"}
{attribute addProperty SizeInBites "34"}
{attribute addProperty SizeInBytes "4.25"}
TYPE EK1501_963BF4D7 :
STRUCT
	{attribute addProperty Name "ID"}
	ID : ID_90FEAF08;
	{attribute addProperty Name "WcState"}
	WcState : WcState_98A4DF75;
	{attribute addProperty Name "InfoData"}
	InfoData : InfoData_192954DE;
END_STRUCT
END_TYPE

// ---- DUTs/IO/Boxes/EK1541_963BF4D7.TcDUT
{attribute addProperty BoxType "EK1541-0000-0016"}
{attribute addProperty Id "IDAT %I*ID_90FEAF081620WcStateAT %I*WcState_98A4DF7520.250InfoDataAT %I*InfoData_192954DE1620"}
{attribute addProperty CRC "1114059904"}
{attribute addProperty SizeInBites "34"}
{attribute addProperty SizeInBytes "4.25"}
TYPE EK1541_963BF4D7 :
STRUCT
	{attribute addProperty Name "ID"}
	ID : ID_90FEAF08;
	{attribute addProperty Name "WcState"}
	WcState : WcState_98A4DF75;
	{attribute addProperty Name "InfoData"}
	InfoData : InfoData_192954DE;
END_STRUCT
END_TYPE

// ---- DUTs/IO/Boxes/EK1561_179A0949.TcDUT
{attribute addProperty BoxType "EK1561-0000-0018"}
{attribute addProperty Id "InfoDataInfoData_192954DE162"}
{attribute addProperty CRC "395970889"}
{attribute addProperty SizeInBites "16"}
{attribute addProperty SizeInBytes "2"}
TYPE EK1561_179A0949 :
STRUCT
	{attribute addProperty Name "InfoData"}
	InfoData : InfoData_192954DE;
END_STRUCT
END_TYPE

// ---- DUTs/IO/Boxes/EK1521_179A0949.TcDUT
{attribute addProperty BoxType "EK1521-0010-0020"}
{attribute addProperty Id "InfoDataInfoData_192954DE162"}
{attribute addProperty CRC "395970889"}
{attribute addProperty SizeInBites "16"}
{attribute addProperty SizeInBytes "2"}
TYPE EK1521_179A0949 :
STRUCT
	{attribute addProperty Name "InfoData"}
	InfoData : InfoData_192954DE;
END_STRUCT
END_TYPE

// ---- DUTs/IO/Boxes/EK1814_97B4DD11.TcDUT
{attribute addProperty BoxType "EK1814-0000-0016"}
{attribute addProperty Id "ChannelAT %I*ARRAY[0..3] OF Channel_E4AEF59E3240Channel_1AT %Q*ARRAY[0..3] OF Channel_7F374EB03240WcStateAT %I*WcState_98A4DF7520.250InfoDataAT %I*InfoData_192954DE1620"}
{attribute addProperty CRC "4250879022"}
{attribute addProperty SizeInBites "82"}
{attribute addProperty SizeInBytes "10.25"}
TYPE EK1814_97B4DD11 :
STRUCT
	{attribute addProperty Name "Channel"}
	Channel : ARRAY[0..3] OF Channel_E4AEF59E;
	{attribute addProperty Name "Channel_1"}
	Channel_1 : ARRAY[0..3] OF Channel_7F374EB0;
	{attribute addProperty Name "WcState"}
	WcState : WcState_98A4DF75;
	{attribute addProperty Name "InfoData"}
	InfoData : InfoData_192954DE;
END_STRUCT
END_TYPE

// ---- DUTs/IO/Boxes/EK1818_5F755A84.TcDUT
{attribute addProperty BoxType "EK1818-0000-0016"}
{attribute addProperty Id "ChannelAT %I*ARRAY[0..7] OF Channel_E4AEF59E6480Channel_1AT %Q*ARRAY[0..3] OF Channel_7F374EB03240WcStateAT %I*WcState_98A4DF7520.250InfoDataAT %I*InfoData_192954DE1620"}
{attribute addProperty CRC "294826719"}
{attribute addProperty SizeInBites "114"}
{attribute addProperty SizeInBytes "14.25"}
TYPE EK1818_5F755A84 :
STRUCT
	{attribute addProperty Name "Channel"}
	Channel : ARRAY[0..7] OF Channel_E4AEF59E;
	{attribute addProperty Name "Channel_1"}
	Channel_1 : ARRAY[0..3] OF Channel_7F374EB0;
	{attribute addProperty Name "WcState"}
	WcState : WcState_98A4DF75;
	{attribute addProperty Name "InfoData"}
	InfoData : InfoData_192954DE;
END_STRUCT
END_TYPE

// ---- DUTs/IO/Boxes/EK1828_A5978B63.TcDUT
{attribute addProperty BoxType "EK1828-0000-0016"}
{attribute addProperty Id "ChannelAT %I*ARRAY[0..3] OF Channel_E4AEF59E3240Channel_1AT %Q*ARRAY[0..7] OF Channel_7F374EB06480WcStateAT %I*WcState_98A4DF7520.250InfoDataAT %I*InfoData_192954DE1620"}
{attribute addProperty CRC "476205506"}
{attribute addProperty SizeInBites "114"}
{attribute addProperty SizeInBytes "14.25"}
TYPE EK1828_A5978B63 :
STRUCT
	{attribute addProperty Name "Channel"}
	Channel : ARRAY[0..3] OF Channel_E4AEF59E;
	{attribute addProperty Name "Channel_1"}
	Channel_1 : ARRAY[0..7] OF Channel_7F374EB0;
	{attribute addProperty Name "WcState"}
	WcState : WcState_98A4DF75;
	{attribute addProperty Name "InfoData"}
	InfoData : InfoData_192954DE;
END_STRUCT
END_TYPE

// ---- DUTs/IO/Boxes/EK1828_A854BE6D.TcDUT
{attribute addProperty BoxType "EK1828-0010-0016"}
{attribute addProperty Id "ChannelAT %Q*ARRAY[0..7] OF Channel_7F374EB06480WcStateAT %I*WcState_28A8677510.1250InfoDataAT %I*InfoData_192954DE1620"}
{attribute addProperty CRC "1482585628"}
{attribute addProperty SizeInBites "81"}
{attribute addProperty SizeInBytes "10.125"}
TYPE EK1828_A854BE6D :
STRUCT
	{attribute addProperty Name "Channel"}
	Channel : ARRAY[0..7] OF Channel_7F374EB0;
	{attribute addProperty Name "WcState"}
	WcState : WcState_28A86775;
	{attribute addProperty Name "InfoData"}
	InfoData : InfoData_192954DE;
END_STRUCT
END_TYPE

// ---- DUTs/IO/Boxes/EKM1101_87969BFD.TcDUT
{attribute addProperty BoxType "EKM1101-0000-0016"}
{attribute addProperty Id "MMS_Device_InputsAT %I*MMS_Device_Inputs_EB48CD741620MMS_Acceleration_StatusAT %I*MMS_Acceleration_Status_2FF1A4723240MMS_Acceleration_X_AxisAT %I*MMS_Acceleration_X_Axis_2EF51F001620MMS_Acceleration_Y_AxisAT %I*MMS_Acceleration_Y_Axis_2EF51F001620MMS_Acceleration_Z_AxisAT %I*MMS_Acceleration_Z_Axis_2EF51F001620MMS_Acceleration_TimestampAT %I*MMS_Acceleration_Timestamp_0B25C1A46480MMS_Voltage_Us_In_InputsAT %I*MMS_Voltage_Us_In_Inputs_BF33E0C16480MMS_Voltage_Up_In_InputsAT %I*MMS_Voltage_Up_In_Inputs_BF33E0C16480MMS_Voltage_Up_Out_InputsAT %I*MMS_Voltage_Up_Out_Inputs_BF33E0C16480MMS_Device_OutputsAT %Q*MMS_Device_Outputs_39C15ABC1620WcStateAT %I*WcState_98A4DF7520.250InfoDataAT %I*InfoData_0BDED7BF144180"}
{attribute addProperty CRC "3393733415"}
{attribute addProperty SizeInBites "514"}
{attribute addProperty SizeInBytes "64.25"}
TYPE EKM1101_87969BFD :
STRUCT
	{attribute addProperty Name "MMS_Device_Inputs"}
	MMS_Device_Inputs : MMS_Device_Inputs_EB48CD74;
	{attribute addProperty Name "MMS_Acceleration_Status"}
	MMS_Acceleration_Status : MMS_Acceleration_Status_2FF1A472;
	{attribute addProperty Name "MMS_Acceleration_X_Axis"}
	MMS_Acceleration_X_Axis : MMS_Acceleration_X_Axis_2EF51F00;
	{attribute addProperty Name "MMS_Acceleration_Y_Axis"}
	MMS_Acceleration_Y_Axis : MMS_Acceleration_Y_Axis_2EF51F00;
	{attribute addProperty Name "MMS_Acceleration_Z_Axis"}
	MMS_Acceleration_Z_Axis : MMS_Acceleration_Z_Axis_2EF51F00;
	{attribute addProperty Name "MMS_Acceleration_Timestamp"}
	MMS_Acceleration_Timestamp : MMS_Acceleration_Timestamp_0B25C1A4;
	{attribute addProperty Name "MMS_Voltage_Us_In_Inputs"}
	MMS_Voltage_Us_In_Inputs : MMS_Voltage_Us_In_Inputs_BF33E0C1;
	{attribute addProperty Name "MMS_Voltage_Up_In_Inputs"}
	MMS_Voltage_Up_In_Inputs : MMS_Voltage_Up_In_Inputs_BF33E0C1;
	{attribute addProperty Name "MMS_Voltage_Up_Out_Inputs"}
	MMS_Voltage_Up_Out_Inputs : MMS_Voltage_Up_Out_Inputs_BF33E0C1;
	{attribute addProperty Name "MMS_Device_Outputs"}
	MMS_Device_Outputs : MMS_Device_Outputs_39C15ABC;
	{attribute addProperty Name "WcState"}
	WcState : WcState_98A4DF75;
	{attribute addProperty Name "InfoData"}
	InfoData : InfoData_0BDED7BF;
END_STRUCT
END_TYPE

// ---- DUTs/IO/Boxes/EK1960_D284ECC6.TcDUT
{attribute addProperty BoxType "EK1960-0000-0019"}
{attribute addProperty Id "Module_1_FSoEModule_1_FSoE_DD00D81F240300Module_2_FSOUTModule_2_FSOUT_3AD10D8E224280Module_3_FSLOGICModule_3_FSLOGIC_3E6251391620WcStateAT %I*WcState_DC9C971540.50InfoDataAT %I*InfoData_BC63D37F80100"}
{attribute addProperty CRC "2754786688"}
{attribute addProperty SizeInBites "564"}
{attribute addProperty SizeInBytes "70.5"}
TYPE EK1960_D284ECC6 :
STRUCT
	{attribute addProperty Name "Module_1_FSoE"}
	Module_1_FSoE : Module_1_FSoE_DD00D81F;
	{attribute addProperty Name "Module_2_FSOUT"}
	Module_2_FSOUT : Module_2_FSOUT_3AD10D8E;
	{attribute addProperty Name "Module_3_FSLOGIC"}
	Module_3_FSLOGIC : Module_3_FSLOGIC_3E625139;
	{attribute addProperty Name "WcState"}
	WcState : WcState_DC9C9715;
	{attribute addProperty Name "InfoData"}
	InfoData : InfoData_BC63D37F;
END_STRUCT
END_TYPE

// ---- DUTs/IO/Boxes/EK1960_858568AC.TcDUT
{attribute addProperty BoxType "EK1960-0000-0021"}
{attribute addProperty Id "Module_1_FSoEModule_1_FSoE_DA01C73E240300Module_2_FSOUTModule_2_FSOUT_9F3624CE192240Module_3_FSLOGICModule_3_FSLOGIC_3E6251391620WcStateAT %I*WcState_DC9C971540.50InfoDataAT %I*InfoData_BC63D37F80100"}
{attribute addProperty CRC "2317899639"}
{attribute addProperty SizeInBites "532"}
{attribute addProperty SizeInBytes "66.5"}
TYPE EK1960_858568AC :
STRUCT
	{attribute addProperty Name "Module_1_FSoE"}
	Module_1_FSoE : Module_1_FSoE_DA01C73E;
	{attribute addProperty Name "Module_2_FSOUT"}
	Module_2_FSOUT : Module_2_FSOUT_9F3624CE;
	{attribute addProperty Name "Module_3_FSLOGIC"}
	Module_3_FSLOGIC : Module_3_FSLOGIC_3E625139;
	{attribute addProperty Name "WcState"}
	WcState : WcState_DC9C9715;
	{attribute addProperty Name "InfoData"}
	InfoData : InfoData_BC63D37F;
END_STRUCT
END_TYPE

// ---- DUTs/IO/Boxes/EK1960_48A2E243.TcDUT
{attribute addProperty BoxType "EK1960-2600-0019"}
{attribute addProperty Id "Module_1_FSoEModule_1_FSoE_DA1FCD51240300Module_2_FSOUTModule_2_FSOUT_3AD10D8E224280Module_3_FSLOGICModule_3_FSLOGIC_3E6251391620WcStateAT %I*WcState_DC9C971540.50InfoDataAT %I*InfoData_BC63D37F80100"}
{attribute addProperty CRC "2308578376"}
{attribute addProperty SizeInBites "564"}
{attribute addProperty SizeInBytes "70.5"}
TYPE EK1960_48A2E243 :
STRUCT
	{attribute addProperty Name "Module_1_FSoE"}
	Module_1_FSoE : Module_1_FSoE_DA1FCD51;
	{attribute addProperty Name "Module_2_FSOUT"}
	Module_2_FSOUT : Module_2_FSOUT_3AD10D8E;
	{attribute addProperty Name "Module_3_FSLOGIC"}
	Module_3_FSLOGIC : Module_3_FSLOGIC_3E625139;
	{attribute addProperty Name "WcState"}
	WcState : WcState_DC9C9715;
	{attribute addProperty Name "InfoData"}
	InfoData : InfoData_BC63D37F;
END_STRUCT
END_TYPE

// ---- DUTs/IO/Boxes/EK1960_3617E9AF.TcDUT
{attribute addProperty BoxType "EK1960-2600-0021"}
{attribute addProperty Id "Module_1_FSoEModule_1_FSoE_1C2EAE46240300Module_2_FSOUTModule_2_FSOUT_3AD10D8E224280Module_3_FSLOGICModule_3_FSLOGIC_3E6251391620WcStateAT %I*WcState_DC9C971540.50InfoDataAT %I*InfoData_BC63D37F80100"}
{attribute addProperty CRC "2592253150"}
{attribute addProperty SizeInBites "564"}
{attribute addProperty SizeInBytes "70.5"}
TYPE EK1960_3617E9AF :
STRUCT
	{attribute addProperty Name "Module_1_FSoE"}
	Module_1_FSoE : Module_1_FSoE_1C2EAE46;
	{attribute addProperty Name "Module_2_FSOUT"}
	Module_2_FSOUT : Module_2_FSOUT_3AD10D8E;
	{attribute addProperty Name "Module_3_FSLOGIC"}
	Module_3_FSLOGIC : Module_3_FSLOGIC_3E625139;
	{attribute addProperty Name "WcState"}
	WcState : WcState_DC9C9715;
	{attribute addProperty Name "InfoData"}
	InfoData : InfoData_BC63D37F;
END_STRUCT
END_TYPE

// ---- DUTs/IO/Devices/SyncUnitTask_B4157F22.TcDUT
{attribute addProperty BoxType "IODEVICETYPE_ETHERCATPROT"}
{attribute addProperty Id "WcStateWcState_28A8677510.1250InfoDataInfoData_BD06A15F6480"}
{attribute addProperty CRC "3021307682"}
{attribute addProperty SizeInBites "65"}
{attribute addProperty SizeInBytes "8.125"}
TYPE SyncUnitTask_B4157F22 :
STRUCT
	{attribute addProperty Name "WcState"}
	WcState : WcState_28A86775;
	{attribute addProperty Name "InfoData"}
	InfoData : InfoData_BD06A15F;
END_STRUCT
END_TYPE

// ---- DUTs/IO/Devices/SyncUnitTasks_5F8F1DD7.TcDUT
{attribute addProperty BoxType ""}
{attribute addProperty Id "unreferencedAT %I*SyncUnitTask_B4157F22658.1250PlcTaskAT %I*SyncUnitTask_B4157F22658.1250"}
{attribute addProperty CRC "1603214807"}
{attribute addProperty SizeInBites "130"}
{attribute addProperty SizeInBytes "16.25"}
TYPE SyncUnitTasks_5F8F1DD7 :
STRUCT
	{attribute addProperty Name "unreferenced"}
	unreferenced : SyncUnitTask_B4157F22;
	{attribute addProperty Name "PlcTask"}
	PlcTask : SyncUnitTask_B4157F22;
END_STRUCT
END_TYPE

// ---- DUTs/IO/Devices/SyncUnits_BBFB8ED4.TcDUT
{attribute addProperty BoxType ""}
{attribute addProperty Id "defaultSyncUnitTasks_5F8F1DD713016.250"}
{attribute addProperty CRC "3153825492"}
{attribute addProperty SizeInBites "130"}
{attribute addProperty SizeInBytes "16.25"}
TYPE SyncUnits_BBFB8ED4 :
STRUCT
	{attribute addProperty Name "default"}
	default : SyncUnitTasks_5F8F1DD7;
END_STRUCT
END_TYPE

// ---- DUTs/IO/Topology/Beckhoff_EJ1xxxEK1122_5D41058A.TcDUT
{attribute addProperty BoxType "EK1122-0000-0018"}
{attribute addProperty Id "Beckhoff_EJ1xxxsub_EK1100EK1100_179A0949162A_0001_EJ1100_0000_0018EJ1100_179A0949162A_0002_EJ1101_0022_0016EJ1101_6969C2248110.125"}
{attribute addProperty CRC "1564542346"}
{attribute addProperty SizeInBites "113"}
{attribute addProperty SizeInBytes "14.125"}
TYPE Beckhoff_EJ1xxxEK1122_5D41058A EXTENDS EK1122_179A0949 :
STRUCT
	{attribute addProperty Name "Beckhoff_EJ1xxxsub_EK1100"}
	Beckhoff_EJ1xxxsub_EK1100 : EK1100_179A0949;
	{attribute addProperty Name "A_0001_EJ1100_0000_0018"}
	A_0001_EJ1100_0000_0018 : EJ1100_179A0949;
	{attribute addProperty Name "A_0002_EJ1101_0022_0016"}
	A_0002_EJ1101_0022_0016 : EJ1101_6969C224;
END_STRUCT
END_TYPE

// ---- DUTs/IO/Topology/Beckhoff_EJ1xxx_BA4DEDCC.TcDUT
{attribute addProperty BoxType "EK1100-0000-0018"}
{attribute addProperty Id "Beckhoff_EJ1xxxEK1122Beckhoff_EJ1xxxEK1122_5D41058A11314.125A_0004_EJ1008_0000_0017EJ1008_772BB4148210.25A_0005_EJ1128_0000_0016EJ1128_772BB4148210.25A_0006_EJ1809_0000_0017EJ1809_248EAA3414618.25A_0007_EJ1819_0000_0017EJ1819_248EAA3414618.25A_0008_EJ1859_0000_0017EJ1859_538B459D14618.25A_0009_EJ1889_0000_0017EJ1889_248EAA3414618.25A_0003_EJ1122_0000_0016EJ1122_179A0949162"}
{attribute addProperty CRC "3125669324"}
{attribute addProperty SizeInBites "877"}
{attribute addProperty SizeInBytes "109.625"}
TYPE Beckhoff_EJ1xxx_BA4DEDCC EXTENDS EK1100_179A0949 :
STRUCT
	{attribute addProperty Name "Beckhoff_EJ1xxxEK1122"}
	Beckhoff_EJ1xxxEK1122 : Beckhoff_EJ1xxxEK1122_5D41058A;
	{attribute addProperty Name "A_0004_EJ1008_0000_0017"}
	A_0004_EJ1008_0000_0017 : EJ1008_772BB414;
	{attribute addProperty Name "A_0005_EJ1128_0000_0016"}
	A_0005_EJ1128_0000_0016 : EJ1128_772BB414;
	{attribute addProperty Name "A_0006_EJ1809_0000_0017"}
	A_0006_EJ1809_0000_0017 : EJ1809_248EAA34;
	{attribute addProperty Name "A_0007_EJ1819_0000_0017"}
	A_0007_EJ1819_0000_0017 : EJ1819_248EAA34;
	{attribute addProperty Name "A_0008_EJ1859_0000_0017"}
	A_0008_EJ1859_0000_0017 : EJ1859_538B459D;
	{attribute addProperty Name "A_0009_EJ1889_0000_0017"}
	A_0009_EJ1889_0000_0017 : EJ1889_248EAA34;
	{attribute addProperty Name "A_0003_EJ1122_0000_0016"}
	A_0003_EJ1122_0000_0016 : EJ1122_179A0949;
END_STRUCT
END_TYPE

// ---- DUTs/IO/Topology/Beckhoff_EJ2xxxEK1122_7BCCD4D9.TcDUT
{attribute addProperty BoxType "EK1122-0000-0018"}
{attribute addProperty Id "Beckhoff_EJ2xxxsub_EK1100EK1100_179A0949162"}
{attribute addProperty CRC "2077021401"}
{attribute addProperty SizeInBites "16"}
{attribute addProperty SizeInBytes "2"}
TYPE Beckhoff_EJ2xxxEK1122_7BCCD4D9 EXTENDS EK1122_179A0949 :
STRUCT
	{attribute addProperty Name "Beckhoff_EJ2xxxsub_EK1100"}
	Beckhoff_EJ2xxxsub_EK1100 : EK1100_179A0949;
END_STRUCT
END_TYPE

// ---- DUTs/IO/Topology/Beckhoff_EJ2xxx_42F4B05B.TcDUT
{attribute addProperty BoxType "EK1100-0000-0018"}
{attribute addProperty Id "Beckhoff_EJ2xxxEK1122Beckhoff_EJ2xxxEK1122_7BCCD4D9162A_0001_EJ2008_0000_0017EJ2008_A854BE6D8110.125A_0002_EJ2008_0000_0018EJ2008_A854BE6D8110.125A_0003_EJ2128_0000_0016EJ2128_A854BE6D8110.125A_0004_EJ2502_0000_0023EJ2502_68F74D5A11314.125A_0005_EJ2502_0000_0024EJ2502_68F74D5A11314.125A_0006_EJ2521_0224_0016EJ2521_A10F5EEB35444.25A_0007_EJ2522_0000_0022EJ2522_58A1BC1F43454.25A_0008_EJ2809_0000_0017EJ2809_859F43D214518.125A_0009_EJ2889_0000_0016EJ2889_859F43D214518.125A_0010_EJ2889_0000_0017EJ2889_859F43D214518.125"}
{attribute addProperty CRC "1123332187"}
{attribute addProperty SizeInBites "1708"}
{attribute addProperty SizeInBytes "213.5"}
TYPE Beckhoff_EJ2xxx_42F4B05B EXTENDS EK1100_179A0949 :
STRUCT
	{attribute addProperty Name "Beckhoff_EJ2xxxEK1122"}
	Beckhoff_EJ2xxxEK1122 : Beckhoff_EJ2xxxEK1122_7BCCD4D9;
	{attribute addProperty Name "A_0001_EJ2008_0000_0017"}
	A_0001_EJ2008_0000_0017 : EJ2008_A854BE6D;
	{attribute addProperty Name "A_0002_EJ2008_0000_0018"}
	A_0002_EJ2008_0000_0018 : EJ2008_A854BE6D;
	{attribute addProperty Name "A_0003_EJ2128_0000_0016"}
	A_0003_EJ2128_0000_0016 : EJ2128_A854BE6D;
	{attribute addProperty Name "A_0004_EJ2502_0000_0023"}
	A_0004_EJ2502_0000_0023 : EJ2502_68F74D5A;
	{attribute addProperty Name "A_0005_EJ2502_0000_0024"}
	A_0005_EJ2502_0000_0024 : EJ2502_68F74D5A;
	{attribute addProperty Name "A_0006_EJ2521_0224_0016"}
	A_0006_EJ2521_0224_0016 : EJ2521_A10F5EEB;
	{attribute addProperty Name "A_0007_EJ2522_0000_0022"}
	A_0007_EJ2522_0000_0022 : EJ2522_58A1BC1F;
	{attribute addProperty Name "A_0008_EJ2809_0000_0017"}
	A_0008_EJ2809_0000_0017 : EJ2809_859F43D2;
	{attribute addProperty Name "A_0009_EJ2889_0000_0016"}
	A_0009_EJ2889_0000_0016 : EJ2889_859F43D2;
	{attribute addProperty Name "A_0010_EJ2889_0000_0017"}
	A_0010_EJ2889_0000_0017 : EJ2889_859F43D2;
END_STRUCT
END_TYPE

// ---- DUTs/IO/Topology/Beckhoff_EJ3xxxEK1122_6922078E.TcDUT
{attribute addProperty BoxType "EK1122-0000-0018"}
{attribute addProperty Id "Beckhoff_EJ3xxxsub_EK1100EK1100_179A0949162"}
{attribute addProperty CRC "1763837838"}
{attribute addProperty SizeInBites "16"}
{attribute addProperty SizeInBytes "2"}
TYPE Beckhoff_EJ3xxxEK1122_6922078E EXTENDS EK1122_179A0949 :
STRUCT
	{attribute addProperty Name "Beckhoff_EJ3xxxsub_EK1100"}
	Beckhoff_EJ3xxxsub_EK1100 : EK1100_179A0949;
END_STRUCT
END_TYPE

// ---- DUTs/IO/Topology/Beckhoff_EJ3xxx_F355313D.TcDUT
{attribute addProperty BoxType "EK1100-0000-0018"}
{attribute addProperty Id "Beckhoff_EJ3xxxEK1122Beckhoff_EJ3xxxEK1122_6922078E162A_0001_EJ3004_0000_0019EJ3004_25122C2021026.25A_0002_EJ3004_0000_0020EJ3004_BB82145621026.25A_0003_EJ3004_0000_0021EJ3004_BB82145621026.25A_0004_EJ3048_0000_0020EJ3048_EA60A07733842.25A_0005_EJ3058_0000_0020EJ3058_EA60A07733842.25A_0006_EJ3068_0000_0020EJ3068_EA60A07733842.25A_0007_EJ3068_0000_0021EJ3068_EA60A07733842.25A_0008_EJ3104_0000_0019EJ3104_B7B5302521026.25A_0009_EJ3104_0000_0020EJ3104_B7B5302521026.25A_0010_EJ3104_0000_0021EJ3104_B7B5302521026.25A_0011_EJ3108_0000_0017EJ3108_EA60A07733842.25A_0012_EJ3108_0000_0018EJ3108_060F55FF33842.25A_0013_EJ3108_0000_0019EJ3108_060F55FF33842.25A_0014_EJ3202_0000_0019EJ3202_559337F514618.25A_0015_EJ3202_0000_0020EJ3202_559337F514618.25A_0016_EJ3202_0000_0021EJ3202_559337F514618.25A_0017_EJ3214_0000_0016EJ3214_712ECA1B21026.25A_0018_EJ3255_0000_0023EJ3255_7B3AD95824230.25A_0019_EJ3318_0000_0017EJ3318_4B9E477A40250.25"}
{attribute addProperty CRC "4082446653"}
{attribute addProperty SizeInBites "4934"}
{attribute addProperty SizeInBytes "616.75"}
TYPE Beckhoff_EJ3xxx_F355313D EXTENDS EK1100_179A0949 :
STRUCT
	{attribute addProperty Name "Beckhoff_EJ3xxxEK1122"}
	Beckhoff_EJ3xxxEK1122 : Beckhoff_EJ3xxxEK1122_6922078E;
	{attribute addProperty Name "A_0001_EJ3004_0000_0019"}
	A_0001_EJ3004_0000_0019 : EJ3004_25122C20;
	{attribute addProperty Name "A_0002_EJ3004_0000_0020"}
	A_0002_EJ3004_0000_0020 : EJ3004_BB821456;
	{attribute addProperty Name "A_0003_EJ3004_0000_0021"}
	A_0003_EJ3004_0000_0021 : EJ3004_BB821456;
	{attribute addProperty Name "A_0004_EJ3048_0000_0020"}
	A_0004_EJ3048_0000_0020 : EJ3048_EA60A077;
	{attribute addProperty Name "A_0005_EJ3058_0000_0020"}
	A_0005_EJ3058_0000_0020 : EJ3058_EA60A077;
	{attribute addProperty Name "A_0006_EJ3068_0000_0020"}
	A_0006_EJ3068_0000_0020 : EJ3068_EA60A077;
	{attribute addProperty Name "A_0007_EJ3068_0000_0021"}
	A_0007_EJ3068_0000_0021 : EJ3068_EA60A077;
	{attribute addProperty Name "A_0008_EJ3104_0000_0019"}
	A_0008_EJ3104_0000_0019 : EJ3104_B7B53025;
	{attribute addProperty Name "A_0009_EJ3104_0000_0020"}
	A_0009_EJ3104_0000_0020 : EJ3104_B7B53025;
	{attribute addProperty Name "A_0010_EJ3104_0000_0021"}
	A_0010_EJ3104_0000_0021 : EJ3104_B7B53025;
	{attribute addProperty Name "A_0011_EJ3108_0000_0017"}
	A_0011_EJ3108_0000_0017 : EJ3108_EA60A077;
	{attribute addProperty Name "A_0012_EJ3108_0000_0018"}
	A_0012_EJ3108_0000_0018 : EJ3108_060F55FF;
	{attribute addProperty Name "A_0013_EJ3108_0000_0019"}
	A_0013_EJ3108_0000_0019 : EJ3108_060F55FF;
	{attribute addProperty Name "A_0014_EJ3202_0000_0019"}
	A_0014_EJ3202_0000_0019 : EJ3202_559337F5;
	{attribute addProperty Name "A_0015_EJ3202_0000_0020"}
	A_0015_EJ3202_0000_0020 : EJ3202_559337F5;
	{attribute addProperty Name "A_0016_EJ3202_0000_0021"}
	A_0016_EJ3202_0000_0021 : EJ3202_559337F5;
	{attribute addProperty Name "A_0017_EJ3214_0000_0016"}
	A_0017_EJ3214_0000_0016 : EJ3214_712ECA1B;
	{attribute addProperty Name "A_0018_EJ3255_0000_0023"}
	A_0018_EJ3255_0000_0023 : EJ3255_7B3AD958;
	{attribute addProperty Name "A_0019_EJ3318_0000_0017"}
	A_0019_EJ3318_0000_0017 : EJ3318_4B9E477A;
END_STRUCT
END_TYPE

// ---- DUTs/IO/Topology/Beckhoff_EJ4xxxEK1122_15AA3F2B.TcDUT
{attribute addProperty BoxType "EK1122-0000-0018"}
{attribute addProperty Id "Beckhoff_EJ4xxxsub_EK1100EK1100_179A0949162"}
{attribute addProperty CRC "363478827"}
{attribute addProperty SizeInBites "16"}
{attribute addProperty SizeInBytes "2"}
TYPE Beckhoff_EJ4xxxEK1122_15AA3F2B EXTENDS EK1122_179A0949 :
STRUCT
	{attribute addProperty Name "Beckhoff_EJ4xxxsub_EK1100"}
	Beckhoff_EJ4xxxsub_EK1100 : EK1100_179A0949;
END_STRUCT
END_TYPE

// ---- DUTs/IO/Topology/Beckhoff_EJ4xxx_B433EAC7.TcDUT
{attribute addProperty BoxType "EK1100-0000-0018"}
{attribute addProperty Id "Beckhoff_EJ4xxxEK1122Beckhoff_EJ4xxxEK1122_15AA3F2B162A_0001_EJ4002_0000_0017EJ4002_19A75BD911314.125A_0002_EJ4002_0000_0018EJ4002_BF483E0111314.125A_0003_EJ4004_0000_0020EJ4004_9786CACB14518.125A_0004_EJ4008_0000_0020EJ4008_D5FA9EBB20926.125A_0005_EJ4018_0000_0016EJ4018_D5FA9EBB20926.125A_0006_EJ4024_0000_0020EJ4024_9786CACB14518.125A_0007_EJ4132_0000_0019EJ4132_19A75BD911314.125A_0008_EJ4134_0000_0019EJ4134_FEE36ED014518.125A_0009_EJ4134_0000_0020EJ4134_FEE36ED014518.125"}
{attribute addProperty CRC "3023301319"}
{attribute addProperty SizeInBites "1353"}
{attribute addProperty SizeInBytes "169.125"}
TYPE Beckhoff_EJ4xxx_B433EAC7 EXTENDS EK1100_179A0949 :
STRUCT
	{attribute addProperty Name "Beckhoff_EJ4xxxEK1122"}
	Beckhoff_EJ4xxxEK1122 : Beckhoff_EJ4xxxEK1122_15AA3F2B;
	{attribute addProperty Name "A_0001_EJ4002_0000_0017"}
	A_0001_EJ4002_0000_0017 : EJ4002_19A75BD9;
	{attribute addProperty Name "A_0002_EJ4002_0000_0018"}
	A_0002_EJ4002_0000_0018 : EJ4002_BF483E01;
	{attribute addProperty Name "A_0003_EJ4004_0000_0020"}
	A_0003_EJ4004_0000_0020 : EJ4004_9786CACB;
	{attribute addProperty Name "A_0004_EJ4008_0000_0020"}
	A_0004_EJ4008_0000_0020 : EJ4008_D5FA9EBB;
	{attribute addProperty Name "A_0005_EJ4018_0000_0016"}
	A_0005_EJ4018_0000_0016 : EJ4018_D5FA9EBB;
	{attribute addProperty Name "A_0006_EJ4024_0000_0020"}
	A_0006_EJ4024_0000_0020 : EJ4024_9786CACB;
	{attribute addProperty Name "A_0007_EJ4132_0000_0019"}
	A_0007_EJ4132_0000_0019 : EJ4132_19A75BD9;
	{attribute addProperty Name "A_0008_EJ4134_0000_0019"}
	A_0008_EJ4134_0000_0019 : EJ4134_FEE36ED0;
	{attribute addProperty Name "A_0009_EJ4134_0000_0020"}
	A_0009_EJ4134_0000_0020 : EJ4134_FEE36ED0;
END_STRUCT
END_TYPE

// ---- DUTs/IO/Topology/Beckhoff_EJ5xxxEK1122_0744EC7C.TcDUT
{attribute addProperty BoxType "EK1122-0000-0018"}
{attribute addProperty Id "Beckhoff_EJ5xxxsub_EK1100EK1100_179A0949162"}
{attribute addProperty CRC "121957500"}
{attribute addProperty SizeInBites "16"}
{attribute addProperty SizeInBytes "2"}
TYPE Beckhoff_EJ5xxxEK1122_0744EC7C EXTENDS EK1122_179A0949 :
STRUCT
	{attribute addProperty Name "Beckhoff_EJ5xxxsub_EK1100"}
	Beckhoff_EJ5xxxsub_EK1100 : EK1100_179A0949;
END_STRUCT
END_TYPE

